// TwinCAT 3 PLC project PLC
// ProgramVersion: 3.1.4024.0
// libraries:
//   EfficientIO Energy Basic, * (EfficientIO)
//   Lynus Persistent Data V1, * (Lynus AG)
//   Lynus Standards, * (EfficientIO)
//   Tc2_EtherCAT, * (Beckhoff Automation GmbH)
//   Tc2_Standard, * (Beckhoff Automation GmbH)
//   Tc2_System, * (Beckhoff Automation GmbH)
//   Tc2_Utilities, * (Beckhoff Automation GmbH)
//   Tc3_Module, * (Beckhoff Automation GmbH)
// project tree:
//   FBs/EL3443_DPM/DUTs/ E_EL3443_DPM_Phase.TcDUT, E_EL3443_DPM_Total.TcDUT, MDP5001_341_7CD731EE.TcDUT (not stored), MDP5001_341_I_7CD731EE.TcDUT (not stored), MDP5001_341_O_7CD731EE.TcDUT (not stored), ST_EL3443_DPM_MUX_REAL.TcDUT (not stored), ST_EL3443_DPM_MUX_ULINT.TcDUT (not stored), ST_EL3443_DPM_StatusLx.TcDUT (not stored), ST_EL3443_DPM_StatusTotal.TcDUT (not stored), ST_EL3443_DPM_VariantLx.TcDUT (not stored), ST_EL3443_DPM_VariantTotal.TcDUT, ST_EL3443_DPM_VariantValues.TcDUT (not stored)
//   FBs/EL3443_DPM/ FB_EL3443_DPM.TcPOU (not stored)
//   FBs/EL3446 FW02 or higher/DUTs/ E_EL3446_Phase.TcDUT (not stored), MDP5001_342_066CA8C6.TcDUT (not stored), MDP5001_342_I_066CA8C6.TcDUT (not stored), MDP5001_342_O_066CA8C6.TcDUT (not stored), ST_EL3446_MUX_REAL.TcDUT (not stored), ST_EL3446_MUX_ULINT.TcDUT (not stored), ST_EL3446_StatusIx.TcDUT (not stored), ST_EL3446_VariantIx.TcDUT (not stored), ST_EL3446_VariantValues.TcDUT (not stored)
//   FBs/EL3446 FW02 or higher/ FB_EL3446.TcPOU (not stored)
//   FBs/ FB_CoE_EL3443.TcPOU, FB_CoE_EL3446.TcPOU (not stored), FB_EM_Beckhoff_EL3443.TcPOU, FB_EM_Beckhoff_EL3446.TcPOU
//   / PlcTask.TcTTO
//   POUs/ prgEM.TcPOU, prgHW.TcPOU
// real-time tasks:
//   TASK PlcTask: cycle T#10ms, priority 20, ADS port 350
// I/O:
//   DEVICE Gerät 2 (EtherCAT), AmsNetId 5.146.127.90.3.1
//     Klemme 1 (EK1200) [EK1200-5000 EtherCAT Netzteil (2A E-Bus)]
//       Klemme 2 (EL3443) [EL3443 3K. Leistungsmessung]
//       Klemme 3 (EL3446) [EL3446 DPM 6 K. Strommessklemme]
//       Klemme 4 (EL9011) [EL9011 Endklemme]
// variable links:
//   PLC/PLC Instance <-> Device 2 (EtherCAT)/Term 1 (EK1200)/Term 2 (EL3443)
//     PlcTask Inputs/prgHW.MDP5001_341_DPM_Data_Data_{1..20} <-> DPM Data/Data {1..20}  (20 links)
//     PlcTask Inputs/prgHW.MDP5001_341_L1_Basic_Current <-> L1 Basic/Current
//     PlcTask Inputs/prgHW.MDP5001_341_L2_Basic_Current <-> L2 Basic/Current
//     PlcTask Inputs/prgHW.MDP5001_341_L3_Basic_Current <-> L3 Basic/Current
//     PlcTask Inputs/prgHW.MDP5001_341_L1_Basic_Voltage <-> L1 Basic/Voltage
//     PlcTask Inputs/prgHW.MDP5001_341_L2_Basic_Voltage <-> L2 Basic/Voltage
//     PlcTask Inputs/prgHW.MDP5001_341_L3_Basic_Voltage <-> L3 Basic/Voltage
//     PlcTask Inputs/prgHW.MDP5001_341_L1_Power_Active_Power <-> L1 Power/Active Power
//     PlcTask Inputs/prgHW.MDP5001_341_L2_Power_Active_Power <-> L2 Power/Active Power
//     PlcTask Inputs/prgHW.MDP5001_341_L3_Power_Active_Power <-> L3 Power/Active Power
//     PlcTask Inputs/prgHW.MDP5001_341_L1_Power_Apparent_Power <-> L1 Power/Apparent Power
//     PlcTask Inputs/prgHW.MDP5001_341_L2_Power_Apparent_Power <-> L2 Power/Apparent Power
//     PlcTask Inputs/prgHW.MDP5001_341_L3_Power_Apparent_Power <-> L3 Power/Apparent Power
//     PlcTask Inputs/prgHW.MDP5001_341_L1_Power_Power_Factor <-> L1 Power/Power Factor
//     PlcTask Inputs/prgHW.MDP5001_341_L2_Power_Power_Factor <-> L2 Power/Power Factor
//     PlcTask Inputs/prgHW.MDP5001_341_L3_Power_Power_Factor <-> L3 Power/Power Factor
//     PlcTask Inputs/prgHW.MDP5001_341_L1_Power_Reactive_Power <-> L1 Power/Reactive Power
//     PlcTask Inputs/prgHW.MDP5001_341_L2_Power_Reactive_Power <-> L2 Power/Reactive Power
//     PlcTask Inputs/prgHW.MDP5001_341_L3_Power_Reactive_Power <-> L3 Power/Reactive Power
//     PlcTask Inputs/prgHW.MDP5001_341_L1_Status_Current_Guard_Error <-> L1 Status/Current Guard Error
//     PlcTask Inputs/prgHW.MDP5001_341_L2_Status_Current_Guard_Error <-> L2 Status/Current Guard Error
//     PlcTask Inputs/prgHW.MDP5001_341_L3_Status_Current_Guard_Error <-> L3 Status/Current Guard Error
//     PlcTask Inputs/prgHW.MDP5001_341_L1_Status_Current_Guard_Warning <-> L1 Status/Current Guard Warning
//     PlcTask Inputs/prgHW.MDP5001_341_L2_Status_Current_Guard_Warning <-> L2 Status/Current Guard Warning
//     PlcTask Inputs/prgHW.MDP5001_341_L3_Status_Current_Guard_Warning <-> L3 Status/Current Guard Warning
//     PlcTask Inputs/prgHW.MDP5001_341_L1_Status_Inaccurate_Current <-> L1 Status/Inaccurate Current
//     PlcTask Inputs/prgHW.MDP5001_341_L2_Status_Inaccurate_Current <-> L2 Status/Inaccurate Current
//     PlcTask Inputs/prgHW.MDP5001_341_L3_Status_Inaccurate_Current <-> L3 Status/Inaccurate Current
//     PlcTask Inputs/prgHW.MDP5001_341_L1_Status_Inaccurate_Voltage <-> L1 Status/Inaccurate Voltage
//     PlcTask Inputs/prgHW.MDP5001_341_L2_Status_Inaccurate_Voltage <-> L2 Status/Inaccurate Voltage
//     PlcTask Inputs/prgHW.MDP5001_341_L3_Status_Inaccurate_Voltage <-> L3 Status/Inaccurate Voltage
//     PlcTask Inputs/prgHW.MDP5001_341_L1_Status_Overcurrent <-> L1 Status/Overcurrent
//     PlcTask Inputs/prgHW.MDP5001_341_L2_Status_Overcurrent <-> L2 Status/Overcurrent
//     PlcTask Inputs/prgHW.MDP5001_341_L3_Status_Overcurrent <-> L3 Status/Overcurrent
//     PlcTask Inputs/prgHW.MDP5001_341_L1_Status_Overvoltage <-> L1 Status/Overvoltage
//     PlcTask Inputs/prgHW.MDP5001_341_L2_Status_Overvoltage <-> L2 Status/Overvoltage
//     PlcTask Inputs/prgHW.MDP5001_341_L3_Status_Overvoltage <-> L3 Status/Overvoltage
//     PlcTask Inputs/prgHW.MDP5001_341_L1_Status_TxPDO_Toggle <-> L1 Status/TxPDO Toggle
//     PlcTask Inputs/prgHW.MDP5001_341_L2_Status_TxPDO_Toggle <-> L2 Status/TxPDO Toggle
//     PlcTask Inputs/prgHW.MDP5001_341_L3_Status_TxPDO_Toggle <-> L3 Status/TxPDO Toggle
//     PlcTask Inputs/prgHW.MDP5001_341_L1_Status_Voltage_Guard_Error <-> L1 Status/Voltage Guard Error
//     PlcTask Inputs/prgHW.MDP5001_341_L2_Status_Voltage_Guard_Error <-> L2 Status/Voltage Guard Error
//     PlcTask Inputs/prgHW.MDP5001_341_L3_Status_Voltage_Guard_Error <-> L3 Status/Voltage Guard Error
//     PlcTask Inputs/prgHW.MDP5001_341_L1_Status_Voltage_Guard_Warning <-> L1 Status/Voltage Guard Warning
//     PlcTask Inputs/prgHW.MDP5001_341_L2_Status_Voltage_Guard_Warning <-> L2 Status/Voltage Guard Warning
//     PlcTask Inputs/prgHW.MDP5001_341_L3_Status_Voltage_Guard_Warning <-> L3 Status/Voltage Guard Warning
//     PlcTask Inputs/prgHW.MDP5001_341_L1_Status_Voltage_Sign_Bit <-> L1 Status/Voltage Sign Bit
//     PlcTask Inputs/prgHW.MDP5001_341_L2_Status_Voltage_Sign_Bit <-> L2 Status/Voltage Sign Bit
//     PlcTask Inputs/prgHW.MDP5001_341_L3_Status_Voltage_Sign_Bit <-> L3 Status/Voltage Sign Bit
//     PlcTask Inputs/prgHW.MDP5001_341_Total_Basic_Calculated_Neutral_Line_Current <-> Total Basic/Calculated Neutral Line Current
//     PlcTask Inputs/prgHW.MDP5001_341_Total_Basic_Frequency <-> Total Basic/Frequency
//     PlcTask Inputs/prgHW.MDP5001_341_Total_Basic_Power_Factor <-> Total Basic/Power Factor
//     PlcTask Inputs/prgHW.MDP5001_341_Total_Status_Active_Power_Guard_Error <-> Total Status/Active Power Guard Error
//     PlcTask Inputs/prgHW.MDP5001_341_Total_Status_Active_Power_Guard_Warning <-> Total Status/Active Power Guard Warning
//     PlcTask Inputs/prgHW.MDP5001_341_Total_Status_Apparent_Power_Guard_Error <-> Total Status/Apparent Power Guard Error
//     PlcTask Inputs/prgHW.MDP5001_341_Total_Status_Apparent_Power_Guard_Warning <-> Total Status/Apparent Power Guard Warning
//     PlcTask Inputs/prgHW.MDP5001_341_Total_Status_Frequency_Guard_Error <-> Total Status/Frequency Guard Error
//     PlcTask Inputs/prgHW.MDP5001_341_Total_Status_Frequency_Guard_Warning <-> Total Status/Frequency Guard Warning
//     PlcTask Inputs/prgHW.MDP5001_341_Total_Status_Grid_Direction <-> Total Status/Grid Direction
//     PlcTask Inputs/prgHW.MDP5001_341_Total_Status_Neutral_Current_Guard_Error <-> Total Status/Neutral Current Guard Error
//     PlcTask Inputs/prgHW.MDP5001_341_Total_Status_Neutral_Current_Guard_Warning <-> Total Status/Neutral Current Guard Warning
//     PlcTask Inputs/prgHW.MDP5001_341_Total_Status_Power_Quality_Factor <-> Total Status/Power Quality Factor
//     PlcTask Inputs/prgHW.MDP5001_341_Total_Status_Power_Quality_Guard_Error <-> Total Status/Power Quality Guard Error
//     PlcTask Inputs/prgHW.MDP5001_341_Total_Status_Power_Quality_Guard_Warning <-> Total Status/Power Quality Guard Warning
//     PlcTask Inputs/prgHW.MDP5001_341_Total_Status_System_State <-> Total Status/System State
//     PlcTask Inputs/prgHW.MDP5001_341_Total_Status_TxPDO_State <-> Total Status/TxPDO State
//     PlcTask Inputs/prgHW.MDP5001_341_Total_Status_TxPDO_Toggle <-> Total Status/TxPDO Toggle
//     PlcTask Inputs/prgHW.MDP5001_341_Total_Variant_Value_In_Index_1_REAL <-> Total Variant Value In/Index 1 REAL
//     PlcTask Inputs/prgHW.MDP5001_341_Total_Variant_Value_In_Index_2_REAL <-> Total Variant Value In/Index 2 REAL
//     PlcTask Inputs/prgHW.MDP5001_341_Total_Variant_Value_In_Index_3_REAL <-> Total Variant Value In/Index 3 REAL
//     PlcTask Inputs/prgHW.MDP5001_341_Total_Variant_Value_In_Index_4_ULINT <-> Total Variant Value In/Index 4 ULINT
//     PlcTask Inputs/prgHW.MDP5001_341_Total_Variant_Value_In_TxPDO_Toggle <-> Total Variant Value In/TxPDO Toggle
//     PlcTask Inputs/prgHW.MDP5001_341_Total_Variant_Value_In_Value_1_REAL <-> Total Variant Value In/Value 1 REAL
//     PlcTask Inputs/prgHW.MDP5001_341_Total_Variant_Value_In_Value_2_REAL <-> Total Variant Value In/Value 2 REAL
//     PlcTask Inputs/prgHW.MDP5001_341_Total_Variant_Value_In_Value_3_REAL <-> Total Variant Value In/Value 3 REAL
//     PlcTask Inputs/prgHW.MDP5001_341_Total_Variant_Value_In_Value_4_ULINT <-> Total Variant Value In/Value 4 ULINT
//     PlcTask Outputs/prgHW.MDP5001_341_Total_Interval_Reset_Interval <-> Total Interval/Reset Interval
//     PlcTask Outputs/prgHW.MDP5001_341_Total_Variant_Value_Out_Index_1_REAL <-> Total Variant Value Out/Index 1 REAL
//     PlcTask Outputs/prgHW.MDP5001_341_Total_Variant_Value_Out_Index_2_REAL <-> Total Variant Value Out/Index 2 REAL
//     PlcTask Outputs/prgHW.MDP5001_341_Total_Variant_Value_Out_Index_3_REAL <-> Total Variant Value Out/Index 3 REAL
//     PlcTask Outputs/prgHW.MDP5001_341_Total_Variant_Value_Out_Index_4_ULINT <-> Total Variant Value Out/Index 4 ULINT
//   PLC/PLC Instance <-> Device 2 (EtherCAT)/Term 1 (EK1200)/Term 3 (EL3446)
//     PlcTask Inputs/prgHW.MDP5001_342_DPM_Variant_Value_In_Index_1_REAL_1 <-> DPM Variant Value In/Index 1 REAL
//     PlcTask Inputs/prgHW.MDP5001_342_DPM_Variant_Value_In_Index_2_REAL_1 <-> DPM Variant Value In/Index 2 REAL
//     PlcTask Inputs/prgHW.MDP5001_342_DPM_Variant_Value_In_Index_3_REAL_1 <-> DPM Variant Value In/Index 3 REAL
//     PlcTask Inputs/prgHW.MDP5001_342_DPM_Variant_Value_In_Index_4_ULINT_1 <-> DPM Variant Value In/Index 4 ULINT
//     PlcTask Inputs/prgHW.MDP5001_342_DPM_Variant_Value_In_TxPDO_Toggle_1 <-> DPM Variant Value In/TxPDO Toggle
//     PlcTask Inputs/prgHW.MDP5001_342_DPM_Variant_Value_In_Value_1_REAL_1 <-> DPM Variant Value In/Value 1 REAL
//     PlcTask Inputs/prgHW.MDP5001_342_DPM_Variant_Value_In_Value_2_REAL_1 <-> DPM Variant Value In/Value 2 REAL
//     PlcTask Inputs/prgHW.MDP5001_342_DPM_Variant_Value_In_Value_3_REAL_1 <-> DPM Variant Value In/Value 3 REAL
//     PlcTask Inputs/prgHW.MDP5001_342_DPM_Variant_Value_In_Value_4_ULINT_1 <-> DPM Variant Value In/Value 4 ULINT
//     PlcTask Inputs/prgHW.MDP5001_342_I{1..6}_Channel_Active_Energy_1 <-> I{1..6} Channel/Active Energy  (6 links)
//     PlcTask Inputs/prgHW.MDP5001_342_I{1..6}_Channel_Active_Power_1 <-> I{1..6} Channel/Active Power  (6 links)
//     PlcTask Inputs/prgHW.MDP5001_342_I{1..6}_Channel_Active_Power_Guard_Error_1 <-> I{1..6} Channel/Active Power Guard Error  (6 links)
//     PlcTask Inputs/prgHW.MDP5001_342_I{1..6}_Channel_Active_Power_Guard_Warning_1 <-> I{1..6} Channel/Active Power Guard Warning  (6 links)
//     PlcTask Inputs/prgHW.MDP5001_342_I{1..6}_Channel_Apparent_Power_1 <-> I{1..6} Channel/Apparent Power  (6 links)
//     PlcTask Inputs/prgHW.MDP5001_342_I{1..6}_Channel_Apparent_Power_Guard_Error_1 <-> I{1..6} Channel/Apparent Power Guard Error  (6 links)
//     PlcTask Inputs/prgHW.MDP5001_342_I{1..6}_Channel_Apparent_Power_Guard_Warning_1 <-> I{1..6} Channel/Apparent Power Guard Warning  (6 links)
//     PlcTask Inputs/prgHW.MDP5001_342_I{1..6}_Channel_Current_1 <-> I{1..6} Channel/Current  (6 links)
//     PlcTask Inputs/prgHW.MDP5001_342_I{1..6}_Channel_Current_Guard_Error_1 <-> I{1..6} Channel/Current Guard Error  (6 links)
//     PlcTask Inputs/prgHW.MDP5001_342_I{1..6}_Channel_Current_Guard_Warning_1 <-> I{1..6} Channel/Current Guard Warning  (6 links)
//     PlcTask Inputs/prgHW.MDP5001_342_I{1..6}_Channel_DPM_Inaccurate_1 <-> I{1..6} Channel/DPM Inaccurate  (6 links)
//     PlcTask Inputs/prgHW.MDP5001_342_I{1..6}_Channel_DPM_Timeout_1 <-> I{1..6} Channel/DPM Timeout  (6 links)
//     PlcTask Inputs/prgHW.MDP5001_342_I{1..6}_Channel_Inaccurate_Current_1 <-> I{1..6} Channel/Inaccurate Current  (6 links)
//     PlcTask Inputs/prgHW.MDP5001_342_I{1..6}_Channel_Overcurrent_1 <-> I{1..6} Channel/Overcurrent  (6 links)
//     PlcTask Inputs/prgHW.MDP5001_342_I{1..6}_Channel_Reactive_Power_Fundamental_1 <-> I{1..6} Channel/Reactive Power Fundamental  (6 links)
//     PlcTask Inputs/prgHW.MDP5001_342_I{1..6}_Channel_Reactive_Power_Guard_Error_1 <-> I{1..6} Channel/Reactive Power Guard Error  (6 links)
//     PlcTask Inputs/prgHW.MDP5001_342_I{1..6}_Channel_Reactive_Power_Guard_Warning_1 <-> I{1..6} Channel/Reactive Power Guard Warning  (6 links)
//     PlcTask Inputs/prgHW.MDP5001_342_I{1..6}_Channel_TxPDO_Toggle_1 <-> I{1..6} Channel/TxPDO Toggle  (6 links)
//     PlcTask Outputs/prgHW.MDP5001_342_DPM_Data_Data_{1..20}_1 <-> DPM Data/Data {1..20}  (20 links)
//     PlcTask Outputs/prgHW.MDP5001_342_DPM_Variant_Value_Out_Index_1_REAL_1 <-> DPM Variant Value Out/Index 1 REAL
//     PlcTask Outputs/prgHW.MDP5001_342_DPM_Variant_Value_Out_Index_2_REAL_1 <-> DPM Variant Value Out/Index 2 REAL
//     PlcTask Outputs/prgHW.MDP5001_342_DPM_Variant_Value_Out_Index_3_REAL_1 <-> DPM Variant Value Out/Index 3 REAL
//     PlcTask Outputs/prgHW.MDP5001_342_DPM_Variant_Value_Out_Index_4_ULINT_1 <-> DPM Variant Value Out/Index 4 ULINT

CONFIGURATION PLC
    RESOURCE PLC ON TwinCAT3
        TASK PlcTask(INTERVAL := T#10ms, PRIORITY := 20);
        PROGRAM prgEM WITH PlcTask : prgEM;
        PROGRAM prgHW WITH PlcTask : prgHW;
    END_RESOURCE
END_CONFIGURATION

// ---- FBs/EL3443_DPM/DUTs/E_EL3443_DPM_Phase.TcDUT
(*This enum is equivalent to the selectors from the documentation " Confirmation of variable output values 1 - 4"*)
{attribute 'qualified_only'}
TYPE E_EL3443_DPM_Phase :
(
    nPhaseL1_OFFSET := 256,      //Offset Channel 1(Phase L1). The offset is added to the base selector     
    nPhaseL2_OFFSET := 512,      //Offset Channel 2(Phase L2). The offset is added to the base selector
    nPhaseL3_OFFSET := 768,      //Offset Channel 3(Phase L3). The offset is added to the base selector
    
    U_RMS := 1,                  // [V] (Real Selector: 1 (Examp.: 257 = 1 + 256 for ch. 1)) RMS value of the voltage
    U_peak := 2,                 // [V] (Real Selector: 2 (Examp.: 770 = 2 + 768 for ch. 3)) Peak value of the instantaneous voltage in the last interval
    U_Last_Zero_Cross := 3,      // [V] (UINT Selector: 3) DC time of the penultimate voltage zero crossing
    U_RMS_Minimum := 4,          // [V] (Real Selector: 4) Minimum RMS value of the voltage in the last interval
    U_RMS_Maximum := 5,          // [V] (Real Selector: 5) Maximum RMS value of the voltage in the last interval
    ULL := 6,                    // [V] (Real Selector: 6) RMS value of the phase-to-phase voltage (Channel 1: U_L1L2; Channel 1: U_L2L3; Channel 3: U_L3L1) 
    I_RMS := 8,                  // [A] (Real Selector: 8) RMS value of the current
    I_peak := 9,                 // [A] (Real Selector: 9) Peak value of the instantaneous current in the last interval
    I_RMS_Minimum := 11,         // [A] (Real Selector: 11) Minimum RMS value of the current in the last interval
    I_RMS_Maximum := 12,         // [A] (Real Selector: 12) Maximum RMS value of the current in the last interval
    Frequency := 17,             // [Hz] (Real Selector: 17) Frequency of this phase
    Phi := 21,                   // [°] (Real Selector: 21) Phase angle of the fundamental wave
    Cos_phi := 22,               // [-] (Real Selector: 22) Cosine of the fundamental wave phase angle
    Power_Factor := 23,          // [-] (Real Selector: 23) Power factor
    P := 26,                     // [W] (Real Selector: 26) Active power
    Pavg := 27,                  // [W] (Real Selector: 27) Average active power during the last interval
    Pmin := 28,                  // [W] (Real Selector: 28) Minimum active power in the last interval
    Pmax := 29,                  // [W] (Real Selector: 29) Maximum active power in the last interval
    S_ := 32,                    // [VA] (Real Selector: 32) Apparent power
    Savg := 33,                  // [VA] (Real Selector: 33) Average apparent power during the last interval
    Smin := 34,                  // [VA] (Real Selector: 34) Minimum apparent power in last interval
    Smax := 35,                  // [VA] (Real Selector: 35) Minimum apparent power in last interval
    Q := 38,                     // [Var] (Real Selector: 38) Reactive power
    Qavg := 39,                  // [Var] (Real Selector: 39) Average reactive power average during the last interval
    Qmin := 40,                  // [Var] (Real Selector: 40) Minimum reactive power in the last interval
    Qmax := 41,                  // [Var] (Real Selector: 41) Maximum reactive power in the last interval
    EP := 45,                    // [mhW] (UINT Selector: 45) Recorded active energy
    EP_pos := 46,                // [mhW] (UINT Selector: 46) Received active energy
    EP_neg := 47,                // [mhW] (UINT Selector: 47) Supplied active energy
	EP_interval := 48, 			// [mhW] (UINT Selector: 48) Recorded active energy in the last interval
	EP_pos_interval := 49, 		// [mhW] (UINT Selector: 49) Received active energy in the last interval
	EP_neg_interval := 50, 		// [mhW] (UINT Selector: 50) Supplied active energy in the last interval
    ES := 51,                    // [mhW] (UINT Selector: 51) Apparent energy
    ES_pos := 52,                // [mhW] (UINT Selector: 52) Apparent energy
    ES_neg := 53,                // [mhW] (UINT Selector: 53) Apparent energy
	ES_interval := 54, 			// [mhW] (UINT Selector: 54) Apparent energy in the last interval
	ES_pos_interval := 55, 		// [mhW] (UINT Selector: 55) Apparent energy in the last interval
	ES_neg_interval := 56, 		// [mhW] (UINT Selector: 56) Apparent energy in the last interval
    EQ_ := 57,                   // [mhW] (UINT Selector: 57) Reactive energy
    EQ_pos := 58,                // [mhW] (UINT Selector: 58) Reactive energy
    EQ_neg := 59,                // [mhW] (UINT Selector: 59) Reactive energy
	EQ_interval := 60, 			// [mhW] (UINT Selector: 60) Reactive energy in the last interval
	EQ_pos_interval := 61, 		// [mhW] (UINT Selector: 62) Reactive energy in the last interval
	EQ_neg_interval := 62, 		// [mhW] (UINT Selector: 63) Reactive energy in the last interval
    THD_U := 95,                 // [-] (Real Selector: 95) "Total Harmonic Distortion" is the distortion factor of the voltage. It indicates the ratio of the harmonic components of an oscillation relative to its fundamental.
    RMS_fund_U := 98,            // [V] (Real Selector: 98) Amplitude of the fundamental wave
    F_Ref_U := 99,               // [Hz] (Real Selector: 99) Reference frequency of the voltage harmonic: Specifies the underlying fundamental frequency, e.g.: 50 or 60 Hz.
    Harmonics_U := 100,          // [% of the fundamental wave] (Real Selector: 100-163) 0 => DC component, 1 => fundamental wave, 2=> 2nd harmonic, 3=> 3rd harmonic
    THD_I := 165,                // [-] (Real Selector: 165) "Total Harmonic Distortion" is the distortion factor of the current. It indicates the ratio of the harmonic components of an oscillation relative to its fundamental.
    TDD_I := 166,                // [% of the maximum current] (Real Selector: 166) "Total Demand Distortion" indicates the ratio between the current harmonics and the maximum current (EL3443: 1A and EL3443-0010: 5A)
    RMS_fund_I := 168,           // [A] (Real Selector: 168) Amplitude of the fundamental wave
    F_Ref_I := 169,              // [Hz] (Real Selector: 169) Reference frequency of the current harmonic: Specifies the underlying fundamental frequency, e.g.: 50 or 60 Hz.
    Harmonics_I := 170,          // [% of the fundamental wave] (Real Selector: 170-233) 0 => DC component, 1 => fundamental wave, 2=> 2nd harmonic, 3=> 3rd harmonic
    Error_INDEX_Not_Valid := 255 // [-] (Real Selector: 255) Error message: The selected index is not available.
)UINT;
END_TYPE

// ---- FBs/EL3443_DPM/DUTs/E_EL3443_DPM_Total.TcDUT
(*This enum is equivalent to the selectors from the documentation " Confirmation of variable output values 1 - 4"*)
{attribute 'qualified_only'}
TYPE E_EL3443_DPM_Total :
(
    nTotal_OFFSET := 1024,           // Offset for total values. The offset is added to the base selector
    
    In_RMS := 8,                     // [A]  (Real Selector: 1032 (= 1024 + 8))  Calculated RMS value of the neutral current
    Power_Factor := 23,              // [-]  (Real Selector: 1047 (= 1024 + 23))  Total power factor over all phases
    Ptot := 26,                      // [W]  (Real Selector: 1050 (= 1024 + 26))  Total active power
    Ptotavg := 27,                   // [W]  (Real Selector: 1051 (= 1024 + 27))  Average total active power during the last interval
    Ptotmin := 28,                   // [W]  (Real Selector: 1052 (= 1024 + 28))  Minimum total active power in the last interval
    Ptotmax := 29,                   // [W]  (Real Selector: 1053 (= 1024 + 29))  Maximum total active power in the last interval
    Stot := 32,                      // [VA]  (Real Selector: 1056 (= 1024 + 32))  Total apparent power
    Stotavg := 33,                   // [VA]  (Real Selector: 1057 (= 1024 + 33))  Average total apparent power during the last interval
    Stotmin := 34,                   // [VA]  (Real Selector: 1058 (= 1024 + 34))  Minimum total apparent power in the last interval
    Stotmax := 35,                   // [VA]  (Real Selector: 1059 (= 1024 + 35))  Maximum total apparent power in the last interval
    Qtot := 38,                      // [Var]  (Real Selector: 1062 (= 1024 + 38))  Total reactive power
    Qtotavg := 39,                   // [Var]  (Real Selector: 1063 (= 1024 + 39))  Average total reactive power during the last interval
    Qtotmin := 40,                   // [Var]  (Real Selector: 1064 (= 1024 + 40))  Minimum total reactive power in the last interval
    Qtotmax := 41,                   // [Var]  (Real Selector: 1065 (= 1024 + 41))  Maximum total reactive power in the last interval
    Eptot := 45,                     // [mWh]  (ULINT Selector: 1069 (= 1024 + 45))  Balanced total active energy
    EPtot_pos := 46,                 // [mWh]  (ULINT Selector: 1070 (= 1024 + 46))  Related total active energy
    EPtot_neg := 47,                 // [mWh]  (ULINT Selector: 1071 (= 1024 + 47))  Input total active energy
    Eptot_interval := 48,            // [mWh]  (ULINT Selector: 1072 (= 1024 + 48))  Balanced total active energy in last interval
    EPtot_pos_interval := 49,        // [mWh]  (ULINT Selector: 1073 (= 1024 + 49))  Total active energy related in the last interval
    EPtot_neg_interval := 50,        // [mWh]  (ULINT Selector: 1074 (= 1024 + 50))  Input total active energy the last interval
    EStot := 51,                     // [mWh]  (ULINT Selector: 1075 (= 1024 + 51))  Total apparent energy
    EStot_pos := 52,                 // [mWh]  (ULINT Selector: 1076 (= 1024 + 52))  Total apparent energy
    EStot_neg := 53,                 // [mWh]  (ULINT Selector: 1077 (= 1024 + 53))  Total apparent energy
    EStot_interval := 54,            // [mWh]  (ULINT Selector: 1078 (= 1024 + 54))  Total apparent energy in the last interval
    EStot_pos_interval := 55,        // [mWh]  (ULINT Selector: 1079 (= 1024 + 55))  Total apparent energy in the last interval
    EStot_neg_interval := 56,        // [mWh]  (ULINT Selector: 1080 (= 1024 + 56))  Total apparent energy in the last interval
    EQtot := 57,                     // [mWh]  (ULINT Selector: 1081 (= 1024 + 57))  Total reactive energy
    EQtot_pos := 58,                 // [mWh]  (ULINT Selector: 1082 (= 1024 + 58))  Total reactive energy
    EQtot_neg := 59,                 // [mWh]  (ULINT Selector: 1083 (= 1024 + 59))  Total reactive energy
    EQtot_interval := 60,            // [mWh]  (ULINT Selector: 1084 (= 1024 + 60))  Total reactive energy in the last interval
    EQtot_pos_interval := 61,        // [mWh]  (ULINT Selector: 1085 (= 1024 + 61))  Total reactive energy in the last interval
    EQtot_neg_interval := 62,        // [mWh]  (ULINT Selector: 1086 (= 1024 + 62))  Total reactive energy in the last interval
    PhiL1L2 := 70,                   // [°]  (Real Selector: 1094 (= 1024 + 70))  Phase shift angle between phase L1 and L2
    PhiL1L3 := 71,                   // [°]  (Real Selector: 1095 (= 1024 + 71))  Phase shift angle between phase L1 and L3
    Unbalance := 72,                 // [-]  (Real Selector: 1096 (= 1024 + 72))  Ratio between negative and positive voltage system
    PQF := 80,                       // [-]  (Real Selector: 1104 (= 1024 + 80))  Power quality factor
    PQF_Avg := 81,                   // [-]  (Real Selector: 1105 (= 1024 + 81))  Average value of the power quality factor during the last interval
    PQF_MIN := 82,                   // [-]  (Real Selector: 1106 (= 1024 + 82))  Minimum power quality factor in the last interval
    PQF_MAX := 83                    // [-]  (Real Selector: 1107 (= 1024 + 83))  Maximum power quality factor in the last interval
)UINT;      
END_TYPE

// ---- FBs/EL3443_DPM/DUTs/ST_EL3443_DPM_VariantTotal.TcDUT
TYPE ST_EL3443_DPM_VariantTotal :
STRUCT
    fIn_RMS : REAL; 			// [A]  (Real Selector: 1032 (= 1024 + 8))  Calculated RMS value of the neutral current
    fPower_Factor : REAL; 		// [-]  (Real Selector: 1047 (= 1024 + 23))  Total power factor over all phases
    fPtot : REAL; 				// [W]  (Real Selector: 1050 (= 1024 + 26))  Total active power
    fPtotavg : REAL; 			// [W]  (Real Selector: 1051 (= 1024 + 27))  Average total active power during the last interval
    fPtotmin : REAL; 			// [W]  (Real Selector: 1052 (= 1024 + 28))  Minimum total active power in the last interval
    fPtotmax : REAL; 			// [W]  (Real Selector: 1053 (= 1024 + 29))  Maximum total active power in the last interval
    fStot : REAL; 				// [VA]  (Real Selector: 1056 (= 1024 + 32))  Total apparent power
    fStotavg : REAL; 			// [VA]  (Real Selector: 1057 (= 1024 + 33))  Average total apparent power during the last interval
    fStotmin : REAL; 			// [VA]  (Real Selector: 1058 (= 1024 + 34))  Minimum total apparent power in the last interval
    fStotmax : REAL; 			// [VA]  (Real Selector: 1059 (= 1024 + 35))  Maximum total apparent power in the last interval
    fQtot : REAL; 				// [Var]  (Real Selector: 1062 (= 1024 + 38))  Total reactive power
    fQtotavg : REAL; 			// [Var]  (Real Selector: 1063 (= 1024 + 39))  Average total reactive power during the last interval
    fQtotmin : REAL; 			// [Var]  (Real Selector: 1064 (= 1024 + 40))  Minimum total reactive power in the last interval
    fQtotmax : REAL; 			// [Var]  (Real Selector: 1065 (= 1024 + 41))  Maximum total reactive power in the last interval
    nEptot : LINT; 				// [mWh]  (LINT Selector: 1069 (= 1024 + 45))  Balanced total active energy
    nEPtot_pos : ULINT; 		// [mWh]  (ULINT Selector: 1070 (= 1024 + 46))  Related total active energy
    nEPtot_neg : ULINT; 		// [mWh]  (ULINT Selector: 1071 (= 1024 + 47))  Input total active energy
    nEptot_interval : LINT; 	// [mWh]  (LINT Selector: 1072 (= 1024 + 48))  Balanced total active energy in last interval
    nEPtot_pos_interval : ULINT;// [mWh]  (ULINT Selector: 1073 (= 1024 + 49))  Total active energy related in the last interval
    nEPtot_neg_interval : ULINT;// [mWh]  (ULINT Selector: 1074 (= 1024 + 50))  Input total active energy the last interval
    nEStot : LINT; 				// [mWh]  (LINT Selector: 1075 (= 1024 + 51))  Total apparent energy
    nEStot_pos : ULINT; 		// [mWh]  (ULINT Selector: 1076 (= 1024 + 52))  Total apparent energy
    nEStot_neg : ULINT; 		// [mWh]  (ULINT Selector: 1077 (= 1024 + 53))  Total apparent energy
    nEStot_interval : LINT; 	// [mWh]  (LINT Selector: 1078 (= 1024 + 54))  Total apparent energy in the last interval
    nEStot_pos_interval : ULINT;// [mWh]  (ULINT Selector: 1079 (= 1024 + 55))  Total apparent energy in the last interval
    nEStot_neg_interval : ULINT;// [mWh]  (ULINT Selector: 1080 (= 1024 + 56))  Total apparent energy in the last interval
    nEQtot : LINT; 				// [mWh]  (LINT Selector: 1081 (= 1024 + 57))  Total reactive energy
    nEQtot_pos : ULINT; 		// [mWh]  (ULINT Selector: 1082 (= 1024 + 58))  Total reactive energy
    nEQtot_neg : ULINT; 		// [mWh]  (ULINT Selector: 1083 (= 1024 + 59))  Total reactive energy
    nEQtot_interval : LINT; 	// [mWh]  (LINT Selector: 1084 (= 1024 + 60))  Total reactive energy in the last interval
    nEQtot_pos_interval : ULINT;// [mWh]  (ULINT Selector: 1085 (= 1024 + 61))  Total reactive energy in the last interval
    nEQtot_neg_interval : ULINT;// [mWh]  (ULINT Selector: 1086 (= 1024 + 62))  Total reactive energy in the last interval
    fPhiL1L2 : REAL; 			// [°]  (Real Selector: 1094 (= 1024 + 70))  Phase shift angle between phase L1 and L2
    fPhiL1L3 : REAL; 			// [°]  (Real Selector: 1095 (= 1024 + 71))  Phase shift angle between phase L1 and L3
    fUnbalance : REAL; 			// [-]  (Real Selector: 1096 (= 1024 + 72))  Ratio between negative and positive voltage system
    fPQF : REAL; 				// [-]  (Real Selector: 1104 (= 1024 + 80))  Power quality factor
    fPQF_Avg : REAL; 			// [-]  (Real Selector: 1105 (= 1024 + 81))  Average value of the power quality factor during the last interval
    fPQF_Min : REAL; 			// [-]  (Real Selector: 1106 (= 1024 + 82))  Minimum power quality factor in the last interval
    fPQF_Max : REAL; 			// [-]  (Real Selector: 1107 (= 1024 + 83))  Maximum power quality factor in the last interval
END_STRUCT
END_TYPE

// ---- POUs/prgEM.TcPOU
PROGRAM prgEM
VAR
	fbEL3443DPM 		: FB_EM_Beckhoff_EL3443;	//EL3443 | PDO Assignment "DPM" (DPM: Distributed Power Measurement) |3-phase power measurement terminal with extended functionality
	fb_EL3446_1			: FB_EM_Beckhoff_EL3446;
	lr_RealPower_Halle	: LREAL;						
	lr_ApparentPower_Halle: LREAL;						
	lr_ReactivePower_Halle: LREAL;						
	lr_Frequency_Halle	: LREAL;						
                                                        
	lr_Voltage_L1N		: LREAL;						
	lr_Voltage_L2N		: LREAL;						
	lr_Voltage_L3N		: LREAL;						
	lr_Voltage_L1L2		: LREAL;						
	lr_Voltage_L2L3		: LREAL;						
	lr_Voltage_L3L1		: LREAL;						
 	lr_Current_L1		: LREAL;						
	lr_Current_L2		: LREAL;						
	lr_Current_L3		: LREAL;						
	lr_Power_House		: LREAL;						
	lr_RealPower_Kran		: LREAL;	
	real_Array_Modbus_Data	AT%MB0 : ARRAY[0..49] OF REAL;

END_VAR
VAR_INPUT
	stEL3443_IO 						: MDP5001_341_7CD731EE;
	stEL3446_IO_1 						: MDP5001_342_066CA8C6; 
	stEL3446_IO_2 						: MDP5001_342_066CA8C6; 
END_VAR
VAR PERSISTENT
	lr_EnergyCounter_Halle	: LREAL;					
END_VAR

// grid measurement
fbEL3443DPM(
	bEnable 	:= TRUE, 
	bInvers_CH1 := FALSE, 
	bInvers_CH2	:= FALSE, 
	bInvers_CH3	:= FALSE, 
	uiCurrentTransformerRatio:= 300,		// two cables,300:1 CTs only over one cable 
	nSlaveAddr 	:= 1001,
	b_SubIndex	:= 2,
	stEL3443_IO := ,
	pDpmData=> , 
	stDataEMPower=> , 
	stDataEMCounter=> , 
	stDataEMPowerRealTime=> , 
	stDataEMCounterRealTime=> );
fbEL3443DPM.stEL3443_IO.MDP5001_341_Input := stEL3443_IO.MDP5001_341_Input;
stEL3443_IO.MDP5001_341_Output	:= fbEL3443DPM.stEL3443_IO.MDP5001_341_Output;
 	
lr_RealPower_Halle		:= fbEL3443DPM.stDataEMPower.lrPowerTotal; 	
lr_ApparentPower_Halle 	:= fbEL3443DPM.stDataEMPower.lrApparentPowerTotal;
lr_ReactivePower_Halle	:= fbEL3443DPM.stDataEMPower.lrReactivePowerTotal;
lr_Frequency_Halle		:= fbEL3443DPM.stDataEMPower.lrFrequency;
lr_Voltage_L1N			:= fbEL3443DPM.stDataEMPower.lrVoltageL1N;
lr_Voltage_L2N			:= fbEL3443DPM.stDataEMPower.lrVoltageL2N;
lr_Voltage_L3N			:= fbEL3443DPM.stDataEMPower.lrVoltageL3N;
lr_Voltage_L1L2			:= fbEL3443DPM.stDataEMPower.lrVoltageL1L2;
lr_Voltage_L2L3			:= fbEL3443DPM.stDataEMPower.lrVoltageL2L3;
lr_Voltage_L3L1			:= fbEL3443DPM.stDataEMPower.lrVoltageL3L1;
lr_EnergyCounter_Halle	:= fbEL3443DPM.stDataEMCounter.lrTotalCounterEnergy_Consumption;
lr_Current_L1			:= fbEL3443DPM.stDataEMPower.lrCurrentL1;
lr_Current_L2			:= fbEL3443DPM.stDataEMPower.lrCurrentL2;
lr_Current_L3			:= fbEL3443DPM.stDataEMPower.lrCurrentL3;
	 
fb_EL3446_1(
	bEnable:= TRUE , 
	bEnableVariantValues:= TRUE, 
	pDpmData:= fbEL3443DPM.pDpmData, 
	nSlaveAddr:= 1002, 
	b_SubIndex	:= 2,
	bInvers_CH1:= FALSE, 
	bInvers_CH2:= FALSE, 
	bInvers_CH3:= FALSE, 
	bInvers_CH4:= FALSE, 
	bInvers_CH5:= FALSE, 
	bInvers_CH6:= FALSE, 
	uiCurrentTransformerRatio_CH1:= 300, 
	uiCurrentTransformerRatio_CH2:= 300, 
	uiCurrentTransformerRatio_CH3:= 300, 
	uiCurrentTransformerRatio_CH4:= 300, 
	uiCurrentTransformerRatio_CH5:= 300, 
	uiCurrentTransformerRatio_CH6:= 300, 
	uiVoltagePhaseSelector_CH1:= , 
	uiVoltagePhaseSelector_CH2:= , 
	uiVoltagePhaseSelector_CH3:= , 
	uiVoltagePhaseSelector_CH4:= , 
	uiVoltagePhaseSelector_CH5:= , 
	uiVoltagePhaseSelector_CH6:= , 
	bEnable3PhaseCH13:= TRUE, 
	bEnable3PhaseCH46:= TRUE, 
	stDataEMPowerRealTime:= fbEL3443DPM.stDataEMPowerRealTime, 
	stEL3446_IO := ,
	stDataEMPower_CH1=> , 
	stDataEMCounter_CH1=> , 
	stDataEMPowerRealTime_CH1=> , 
	stDataEMCounterRealTime_CH1=> , 
	stDataEMPower_CH2=> , 
	stDataEMCounter_CH2=> , 
	stDataEMPowerRealTime_CH2=> , 
	stDataEMCounterRealTime_CH2=> , 
	stDataEMPower_CH3=> , 
	stDataEMCounter_CH3=> , 
	stDataEMPowerRealTime_CH3=> , 
	stDataEMCounterRealTime_CH3=> , 
	stDataEMPower_CH4=> , 
	stDataEMCounter_CH4=> , 
	stDataEMPowerRealTime_CH4=> , 
	stDataEMCounterRealTime_CH4=> , 
	stDataEMPower_CH5=> , 
	stDataEMCounter_CH5=> , 
	stDataEMPowerRealTime_CH5=> , 
	stDataEMCounterRealTime_CH5=> , 
	stDataEMPower_CH6=> , 
	stDataEMCounter_CH6=> , 
	stDataEMPowerRealTime_CH6=> , 
	stDataEMCounterRealTime_CH6=> );
fb_EL3446_1.stEL3446_IO.MDP5001_342_Input := stEL3446_IO_1.MDP5001_342_Input;
stEL3446_IO_1.MDP5001_342_Output := 	fb_EL3446_1.stEL3446_IO.MDP5001_342_Output;

lr_RealPower_Kran := fb_EL3446_1.stDataEMPower_CH1.lrPowerConsumption;

real_Array_Modbus_Data[0] 	:= 		INT_TO_REAL(REAL_TO_INT(LREAL_TO_REAL(lr_RealPower_Halle    *10)))/10 ;
real_Array_Modbus_Data[1] 	:= 		INT_TO_REAL(REAL_TO_INT(LREAL_TO_REAL(lr_ApparentPower_Halle*10)))/10 ;
real_Array_Modbus_Data[2] 	:= 		INT_TO_REAL(REAL_TO_INT(LREAL_TO_REAL(lr_ReactivePower_Halle*10)))/10 ;
real_Array_Modbus_Data[3] 	:= 		INT_TO_REAL(REAL_TO_INT(LREAL_TO_REAL(lr_Frequency_Halle    *10)))/10 ;
real_Array_Modbus_Data[4] 	:= 		INT_TO_REAL(REAL_TO_INT(LREAL_TO_REAL(lr_Voltage_L1N     	*10)))/10 ;
real_Array_Modbus_Data[5] 	:= 		INT_TO_REAL(REAL_TO_INT(LREAL_TO_REAL(lr_Voltage_L2N     	*10)))/10 ;
real_Array_Modbus_Data[6] 	:= 		INT_TO_REAL(REAL_TO_INT(LREAL_TO_REAL(lr_Voltage_L3N    	*10)))/10 ;
real_Array_Modbus_Data[7]	:=      INT_TO_REAL(REAL_TO_INT(LREAL_TO_REAL(lr_Voltage_L1L2		*10)))/10  ;
real_Array_Modbus_Data[8]	:=      INT_TO_REAL(REAL_TO_INT(LREAL_TO_REAL(lr_Voltage_L2L3		*10)))/10  ;
real_Array_Modbus_Data[9]	:=      INT_TO_REAL(REAL_TO_INT(LREAL_TO_REAL(lr_Voltage_L3L1		*10)))/10  ;
real_Array_Modbus_Data[10]	:=      INT_TO_REAL(REAL_TO_INT(LREAL_TO_REAL(lr_Current_L1		  	*10)))/10      ;
real_Array_Modbus_Data[11]	:=      INT_TO_REAL(REAL_TO_INT(LREAL_TO_REAL(lr_Current_L2		  	*10)))/10      ;
real_Array_Modbus_Data[12]	:=      INT_TO_REAL(REAL_TO_INT(LREAL_TO_REAL(lr_Current_L3		  	*10)))/10      ;
real_Array_Modbus_Data[13]	:=      INT_TO_REAL(REAL_TO_INT(LREAL_TO_REAL(lr_RealPower_Kran 	*10)))/10    ;

END_PROGRAM

// ---- FBs/FB_EM_Beckhoff_EL3443.TcPOU
FUNCTION_BLOCK FB_EM_Beckhoff_EL3443
VAR_INPUT
	bEnable							: BOOL;											//Enable the function
 	bInvers_CH1						: BOOL;											//Invert the Output data from Channel 1 
	bInvers_CH2						: BOOL;											//Invert the Output data from Channel 2 
	bInvers_CH3						: BOOL;											//Invert the Output data from Channel 3
	uiCurrentTransformerRatio		: UINT;											//Current Transformer Ratio  
	nSlaveAddr						: UINT;											//EtherCat Slave ID	
 	b_SubIndex						: BYTE;											//AmsNet ID Index, typically 2 or 3
	stEL3443_IO 						: MDP5001_341_7CD731EE;
END_VAR
VAR_OUTPUT
   	pDpmData 						: POINTER TO ARRAY[1..20] OF UDINT;
	stDataEMPower					: ST_ElectricMeter_Output_Power;				//Output structure with Data from Electric Meter (Power Data) 
	stDataEMCounter					: ST_ElectricMeter_Output_Counter;				//Output structure with Data from Electric Meter (Counter Data) 
	stDataEMPowerRealTime			: ST_ElectricMeter_Output_Power;				//Output structure with Data from Electric Meter (Power Data RealTime)
	stDataEMCounterRealTime			: ST_ElectricMeter_Output_Counter;				//Output structure with Data from Electric Meter (Counter Data RealTime) 
END_VAR
VAR
	fbEM							: FB_ElectricMeter;								//Electric Meter Function
	fbEnergyCounter					: FB_EnergyCounter;								//FB energy Counter, because the KL3403 has no nice logic for the Energy value
	fbEL3443DPM 					: FB_EL3443_DPM;
	
	fb_WriteCOE_EL3443	:FB_Coe_EL3443;	
	m_COE_Done: BOOL;
	uiCurrentTransformerRatio_old		: UINT;											//Current Transformer Ratio  
	f_trig_Busy: f_trig;

	
	timDissableFunctions			: TON;											//Timer to dissable the Function after Lynus_Standards.Constants_General.tTimeDissableLynusFunctions Days without connection to the Lynus Cloud
	timResetConnectionOnGVL			: TON;											//Timer to try reset the connection Flag on the GVL. (When somebody delete the Connection Function and make only a onlinechange)
	timSetCounterValues				: TON;											//Timer to set the counter values from the KL3403 Function to the EM Function
	arrPD							: ARRAY[1..7] OF FB_PersistentData_Number;		//Function to save persistent data
	byWaitInStep					: BYTE;											//Wait in Step before start to clean data on PLC
	iStateGVLData					: INT;											//State machine to handle the data on the GVL
	diCounterForGVL					: DINT;											//Counter to clean old data on GVL
	real_Multiplier_CH1: REAL;
	real_Multiplier_CH2: REAL;
	real_Multiplier_CH3: REAL;
END_VAR

//Creator : Stefan Lackner
//Company : EfficientIO
//Date : xx.09.2023
//Version : 1.0.0.0


//With this function is possible to read out all Information from a EL3446

//NOTE for diNr.....Designation => 
//_IN = Here Data come in from other Functions or go out to other functions about the GVL
//_OUT = Here Data go out to other functions about the GVL



(*-------------------------------------------------------------Service from Backend is ready and check the connection to backen for dissabel/enable Function---------------------------------------------------------------*)

//Try to reset the variable for connection on the GVL. When all is normal then the Lynus Mqtt connection function set this variable to true in the next cycle
//When we have no connection to the backend then after Lynus_Standards.Constants_General.tTimeDissableLynusFunctions days the Function is dissabled with all of his functionalities
timResetConnectionOnGVL(IN:= NOT timResetConnectionOnGVL.Q, PT:= T#1H, Q=> , ET=> );
IF timResetConnectionOnGVL.Q THEN 
	Lynus_Standards.GVL_Communicator.bStateConnectionToEnableFunctions := FALSE; 
END_IF
IF NOT Lynus_Standards.GVL_Communicator.bStateConnectionToEnableFunctions THEN 
	timDissableFunctions.IN := TRUE; 
ELSE 
	timDissableFunctions.IN := FALSE; 
END_IF  
timDissableFunctions(IN:= , PT:= Lynus_Standards.Constants_General.tTimeDissableLynusFunctions, Q=> , ET=> );

// limit inputs
uiCurrentTransformerRatio	 := LIMIT (1,uiCurrentTransformerRatio,10000);


(*----------------------------------------------------------------------------------------EL3446 Communication----------------------------------------------------------------------------------------------*)
// write CoE values for phase selector

IF 	NOT m_COE_Done OR 	uiCurrentTransformerRatio <> uiCurrentTransformerRatio_old THEN
	fb_WriteCOE_EL3443.m_start := TRUE;
	m_COE_Done := TRUE;
	 uiCurrentTransformerRatio_old := uiCurrentTransformerRatio;
END_IF
f_trig_Busy(CLK := fb_WriteCOE_EL3443.m_Busy );
IF f_trig_Busy.Q AND (fb_WriteCOE_EL3443.m_CoE_Write_done OR fb_WriteCOE_EL3443.m_Error) THEN 
	fb_WriteCOE_EL3443.m_start := FALSE;
END_IF

fb_WriteCOE_EL3443(
	m_start:= , 
	nSlaveAddr:= nSlaveAddr, 
	b_SubIndex:= b_SubIndex,
	uiCurrentTransformerRatio:= uiCurrentTransformerRatio, 
	m_Busy=> , 
	m_CoE_Write_done=> , 
	m_Error=> , 
	udint_GetAMSNetID_Error=> , 
	udint_WriteCoE_Error=> );



fbEL3443DPM(
	bEnable:= TRUE, 
	stEL3443_IO:= stEL3443_IO , 
	stStatusTotal=> , 
	stStatusPhase_L1=> , 
	stStatusPhase_L2=> , 
	stStatusPhase_L3=> , 
	stVariantValues=> , 
	pDpmData=> pDpmData, 
	bError=> );






//Invert the Output data, because it is possible that the current transformers have been mounted in different mounting positions.
IF NOT bInvers_CH1 THEN
	real_Multiplier_CH1 := 1;
ELSE
	real_Multiplier_CH1 := -1;
END_IF
IF NOT bInvers_CH2 THEN
	real_Multiplier_CH2 := 1;
ELSE
	real_Multiplier_CH2 := -1;
END_IF
IF NOT bInvers_CH3 THEN
	real_Multiplier_CH3 := 1;
ELSE
	real_Multiplier_CH3 := -1;
END_IF


//Function
fbEM(
	bEnable:= bEnable, 
	bError:= , 
	bEnableReadOutFunction:= FALSE, 
	bWriteWithDelay:= TRUE, 
	bPowerDataInvers:= FALSE,
	bReadOutDataDone:= timSetCounterValues.Q,
	iTimeReadOutInterval:= 0, 
	iErrorCode:= , 
	iWarningCode:= , 
	lrTotalCounterEnergy_Consumption:= fbEnergyCounter.lrTotalCounterEnergy_Consumption,
	lrTotalCounterEnergy_Production:= fbEnergyCounter.lrTotalCounterEnergy_Production, 
	lrCounterEnergyT1_Consumption:= fbEnergyCounter.lrCounterEnergyT1_Consumption,
	lrCounterEnergyT2_Consumption:= fbEnergyCounter.lrCounterEnergyT2_Consumption,
	lrCounterEnergyT1_Production:= fbEnergyCounter.lrCounterEnergyT1_Production, 
	lrCounterEnergyT2_Production:= fbEnergyCounter.lrCounterEnergyT2_Production, 
	lrCurrentL1:=  REAL_TO_LREAL(fbEL3443DPM.stEL3443_IO.MDP5001_341_Input.MDP5001_341_L1_Basic_Current ),
	lrVoltageL1N:= REAL_TO_LREAL(fbEL3443DPM.stEL3443_IO.MDP5001_341_Input.MDP5001_341_L1_Basic_Voltage), 
	lrVoltageL1L2:= REAL_TO_LREAL(fbEL3443DPM.stEL3443_IO.MDP5001_341_Input.MDP5001_341_L1_Basic_Voltage * 1.73), 
	lrPowerL1:= REAL_TO_LREAL(fbEL3443DPM.stEL3443_IO.MDP5001_341_Input.MDP5001_341_L1_Power_Active_Power * real_Multiplier_CH1), 
	lrCurrentL2:=  REAL_TO_LREAL(fbEL3443DPM.stEL3443_IO.MDP5001_341_Input.MDP5001_341_L2_Basic_Current),
	lrVoltageL2N:= REAL_TO_LREAL(fbEL3443DPM.stEL3443_IO.MDP5001_341_Input.MDP5001_341_L2_Basic_Voltage), 
	lrVoltageL2L3:= REAL_TO_LREAL(fbEL3443DPM.stEL3443_IO.MDP5001_341_Input.MDP5001_341_L2_Basic_Voltage * 1.73), 
	lrPowerL2:= REAL_TO_LREAL(fbEL3443DPM.stEL3443_IO.MDP5001_341_Input.MDP5001_341_L2_Power_Active_Power  * real_Multiplier_CH2),	
	lrCurrentL3:=  REAL_TO_LREAL(fbEL3443DPM.stEL3443_IO.MDP5001_341_Input.MDP5001_341_L3_Basic_Current),
	lrVoltageL3N:= REAL_TO_LREAL(fbEL3443DPM.stEL3443_IO.MDP5001_341_Input.MDP5001_341_L3_Basic_Voltage), 
	lrVoltageL3L1:= REAL_TO_LREAL(fbEL3443DPM.stEL3443_IO.MDP5001_341_Input.MDP5001_341_L3_Basic_Voltage * 1.73), 
	lrPowerL3:= REAL_TO_LREAL(fbEL3443DPM.stEL3443_IO.MDP5001_341_Input.MDP5001_341_L3_Power_Active_Power * real_Multiplier_CH3),	

	lrPowerTotal:= fbEM.lrPowerL1+fbEM.lrPowerL2+fbEM.lrPowerL3, 
	lrFrequency:= REAL_TO_LREAL(fbEL3443DPM.stEL3443_IO.MDP5001_341_Input.MDP5001_341_Total_Basic_Frequency), 
 	lrApparentPowerTotal:= REAL_TO_LREAL(fbEL3443DPM.stEL3443_IO.MDP5001_341_Input.MDP5001_341_L1_Power_Apparent_Power + fbEL3443DPM.stEL3443_IO.MDP5001_341_Input.MDP5001_341_L2_Power_Apparent_Power + fbEL3443DPM.stEL3443_IO.MDP5001_341_Input.MDP5001_341_L3_Power_Apparent_Power) ,
	lrReactivePowerTotal:= REAL_TO_LREAL(fbEL3443DPM.stEL3443_IO.MDP5001_341_Input.MDP5001_341_L1_Power_Reactive_Power + fbEL3443DPM.stEL3443_IO.MDP5001_341_Input.MDP5001_341_L2_Power_Reactive_Power + fbEL3443DPM.stEL3443_IO.MDP5001_341_Input.MDP5001_341_L3_Power_Reactive_Power) , 
	tTimDelayOutput:= T#5S, 
	stDataEMOutPower=> stDataEMPowerRealTime, 
	stDataEMOutPowerDelay=> stDataEMPower, 
	stDataEMOutCounter=> stDataEMCounterRealTime,
	stDataEMOutCounterDelay=> stDataEMCounter,
	bReadOutMeter=> );
(*----------------------------------------------------------------------------------------Energy Counter Function----------------------------------------------------------------------------------------------*)

fbEnergyCounter(
	byActiveTariff:= 1, 
	lrPowerInput:= (fbEM.lrPowerTotal) / 1000, 
	lrTotalCounterEnergy_Consumption=> , 
	lrTotalCounterEnergy_Production=> , 
	lrCounterEnergyT1_Consumption=> , 
	lrCounterEnergyT2_Consumption=> , 
	lrCounterEnergyT1_Production=> , 
	lrCounterEnergyT2_Production=> );
(*----------------------------------------------------------------------------------------Electric Meter Function----------------------------------------------------------------------------------------------*)

//Error
IF timDissableFunctions.Q THEN 
	fbEM.bWarning := TRUE; 
	fbEM.iWarningCode := 0; 
ELSE 
	fbEM.bWarning := FALSE; 
END_IF 
IF Lynus_Standards.GVL_Energy.stNumberOfDevices.diNumberOfElectricMeters > Constants_Energy.diMaxNumberOfElectricMeters THEN 
	fbEM.bError := TRUE; 
ELSE 
	fbEM.bError := FALSE; 
END_IF
IF Lynus_Standards.GVL_Energy.stNumberOfDevices.diNumberOfElectricMeters > Constants_Energy.diMaxNumberOfElectricMeters THEN 
	fbEM.iErrorCode := 1;
ELSE 
	fbEM.iErrorCode := 0;
END_IF

timSetCounterValues(IN:= bEnable AND NOT timSetCounterValues.Q, PT:= T#2S, Q=> , ET=> );

END_FUNCTION_BLOCK

// ---- FBs/FB_CoE_EL3443.TcPOU
FUNCTION_BLOCK FB_CoE_EL3443
VAR_INPUT
	m_start: BOOL;
	nSlaveAddr	:UINT;
	b_SubIndex	:BYTE;
	uiCurrentTransformerRatio		: UINT;											//CT Ratio
END_VAR
VAR_OUTPUT
	m_Busy: BOOL;
	m_CoE_Write_done: BOOL;
	m_Error: bool;
	udint_GetAMSNetID_Error: UDINT;
	udint_WriteCoE_Error: UDINT;
END_VAR
VAR
	i_State	:UINT:=1;
	fb_GetAMSNetID	:FB_GetLocalAmsNetId;
  	fb_coe_write          : FB_EcCoESdoWrite; // Function Block for writing in CoE


	r_trig_Start: R_trig;
	i_errorCount: INT;
	i_AMSNetID_ReadOut_Succesfull: INT;
	str_AMSNetID: STRING(30);
 	real_Value     : REAL ; (* variable to be written to the CoE Object *)
 	
	i_CoE_Write_Succesfull: INT;

	real_Current_Min_Warning 	: REAL	:=-100;
	real_Current_Min_Error 		: REAL	:=-120;
	real_Current_Max_Warning 	: REAL	:= 100;
	real_Current_Max_Error 		: REAL	:= 120;
	


END_VAR


r_trig_Start(Clk := m_start);
b_SubIndex := LIMIT (1,b_SubIndex,8);
CASE i_State OF
	1: 		// wait for start
	IF r_trig_Start.Q THEN
		i_State := i_State+1;
		m_CoE_Write_done := FALSE;
		m_Busy := TRUE;
		m_Error := FALSE;
	END_IF

	2:		// read out ams net ID	
	fb_GetAMSNetID.bExecute := TRUE;
	i_State := i_State+1;
	
	3: 		// wait for read out
	IF fb_GetAMSNetID.bBusy = FALSE AND NOT fb_GetAMSNetID.bError = TRUE THEN
		fb_GetAMSNetID.bExecute := FALSE;
		i_AMSNetID_ReadOut_Succesfull := i_AMSNetID_ReadOut_Succesfull+1;
		i_State := i_State+1;
	ELSIF fb_GetAMSNetID.bError = TRUE THEN
		fb_GetAMSNetID.bExecute := FALSE;
		i_State := 100;
	END_IF
	
	4: 		// read out AMS Net ID done, convert received data
	str_AMSNetID := concat(BYTE_TO_STRING(fb_GetAMSNetID.AddrBytes[0]),'.');
	str_AMSNetID := concat(str_AMSNetID,BYTE_TO_STRING(fb_GetAMSNetID.AddrBytes[1]));
	str_AMSNetID := concat(str_AMSNetID,'.');	
	str_AMSNetID := concat(str_AMSNetID,BYTE_TO_STRING(fb_GetAMSNetID.AddrBytes[2]));
	str_AMSNetID := concat(str_AMSNetID,'.');
	str_AMSNetID := concat(str_AMSNetID,BYTE_TO_STRING(fb_GetAMSNetID.AddrBytes[3]));
	str_AMSNetID := concat(str_AMSNetID,'.');
	str_AMSNetID := concat(str_AMSNetID,BYTE_TO_STRING(b_SubIndex));
	str_AMSNetID := concat(str_AMSNetID,'.1');
	
	i_State := 10;

	10: 	// write channel 1 
	fb_coe_write.bExecute 	:= TRUE;
	fb_coe_write.nIndex		:= 16#8000;
	fb_coe_write.nSubIndex	:= 16#12; 
	real_Value 			:= UINT_TO_REAL(uiCurrentTransformerRatio);
	fb_coe_write.pSrcBuf	:= ADR(real_Value);
	fb_coe_write.cbBufLen	:= SIZEOF(real_Value);
	i_State := i_State+1;
	
	11: 	// wait for done or error
	IF NOT fb_coe_write.bBusy AND NOT fb_coe_write.bError THEN
		fb_coe_write.bExecute 	:= FALSE;
		i_CoE_Write_Succesfull := i_CoE_Write_Succesfull+1;
		i_State := i_State+1;
	ELSIF fb_coe_write.bError THEN
		fb_coe_write.bExecute 	:= FALSE;
		i_State := 100;
	END_IF

	12:		// wait 
	i_State := 20;
	
	20: 	// write channel 2 
	fb_coe_write.bExecute 	:= TRUE;
	fb_coe_write.nIndex		:= 16#8010;
	fb_coe_write.nSubIndex	:= 16#12; 
	real_Value 			:= UINT_TO_REAL(uiCurrentTransformerRatio);
	fb_coe_write.pSrcBuf	:= ADR(real_Value);
	fb_coe_write.cbBufLen	:= SIZEOF(real_Value);
	i_State := i_State+1;
	
	21: 	// wait for done or error
	IF NOT fb_coe_write.bBusy AND NOT fb_coe_write.bError THEN
		fb_coe_write.bExecute 	:= FALSE;
		i_CoE_Write_Succesfull := i_CoE_Write_Succesfull+1;
		i_State := i_State+1;
	ELSIF fb_coe_write.bError THEN
		fb_coe_write.bExecute 	:= FALSE;
		i_State := 100;
	END_IF

	22:		// wait 
	i_State := 30;

	30: 	// write channel 3 
	fb_coe_write.bExecute 	:= TRUE;
	fb_coe_write.nIndex		:= 16#8020;
	fb_coe_write.nSubIndex	:= 16#12; 
	real_Value 			:= UINT_TO_REAL(uiCurrentTransformerRatio);
	fb_coe_write.pSrcBuf	:= ADR(real_Value);
	fb_coe_write.cbBufLen	:= SIZEOF(real_Value);
	i_State := i_State+1;
	
	31: 	// wait for done or error
	IF NOT fb_coe_write.bBusy AND NOT fb_coe_write.bError THEN
		fb_coe_write.bExecute 	:= FALSE;
		i_CoE_Write_Succesfull := i_CoE_Write_Succesfull+1;
		i_State := i_State+1;
	ELSIF fb_coe_write.bError THEN
		fb_coe_write.bExecute 	:= FALSE;
		i_State := 100;
	END_IF

	32:		// wait 
	i_State := 40;		

	40: 	// write Channel 1 current guard min error 
	fb_coe_write.bExecute 	:= TRUE;
	fb_coe_write.nIndex		:= 16#8001;
	fb_coe_write.nSubIndex	:= 16#15; 
	real_Value 			:= (real_Current_Min_Error);
	fb_coe_write.pSrcBuf	:= ADR(real_Value);
	fb_coe_write.cbBufLen	:= SIZEOF(real_Value);
	i_State := i_State+1;
	
	41: 	// wait for done or error
	IF NOT fb_coe_write.bBusy AND NOT fb_coe_write.bError THEN
		fb_coe_write.bExecute 	:= FALSE;
		i_CoE_Write_Succesfull := i_CoE_Write_Succesfull+1;
		i_State := i_State+1;
	ELSIF fb_coe_write.bError THEN
		fb_coe_write.bExecute 	:= FALSE;
		i_State := 100;
	END_IF
	
	42:		// wait 
	i_State := i_State+1;		

	43: 	// write Channel 1 current guard min warning 
	fb_coe_write.bExecute 	:= TRUE;
	fb_coe_write.nIndex		:= 16#8001;
	fb_coe_write.nSubIndex	:= 16#16; 
	real_Value 			:= (real_Current_Min_Warning);
	fb_coe_write.pSrcBuf	:= ADR(real_Value);
	fb_coe_write.cbBufLen	:= SIZEOF(real_Value);
	i_State := i_State+1;
	
	44: 	// wait for done or error
	IF NOT fb_coe_write.bBusy AND NOT fb_coe_write.bError THEN
		fb_coe_write.bExecute 	:= FALSE;
		i_CoE_Write_Succesfull := i_CoE_Write_Succesfull+1;
		i_State := i_State+1;
	ELSIF fb_coe_write.bError THEN
		fb_coe_write.bExecute 	:= FALSE;
		i_State := 100;
	END_IF

	45:		// wait 
	i_State := i_State+1;		

	46: 	// write Channel 1 current guard max warning 
	fb_coe_write.bExecute 	:= TRUE;
	fb_coe_write.nIndex		:= 16#8001;
	fb_coe_write.nSubIndex	:= 16#17; 
	real_Value 			:= (real_Current_Max_Warning);
	fb_coe_write.pSrcBuf	:= ADR(real_Value);
	fb_coe_write.cbBufLen	:= SIZEOF(real_Value);
	i_State := i_State+1;
	
	47: 	// wait for done or error
	IF NOT fb_coe_write.bBusy AND NOT fb_coe_write.bError THEN
		fb_coe_write.bExecute 	:= FALSE;
		i_CoE_Write_Succesfull := i_CoE_Write_Succesfull+1;
		i_State := i_State+1;
	ELSIF fb_coe_write.bError THEN
		fb_coe_write.bExecute 	:= FALSE;
		i_State := 100;
	END_IF
	
	48:		// wait 
	i_State := i_State+1;		

	49: 	// write Channel 1 current guard max error 
	fb_coe_write.bExecute 	:= TRUE;
	fb_coe_write.nIndex		:= 16#8001;
	fb_coe_write.nSubIndex	:= 16#18; 
	real_Value 			:= (real_Current_Max_Error);
	fb_coe_write.pSrcBuf	:= ADR(real_Value);
	fb_coe_write.cbBufLen	:= SIZEOF(real_Value);
	i_State := i_State+1;
	
	50: 	// wait for done or error
	IF NOT fb_coe_write.bBusy AND NOT fb_coe_write.bError THEN
		fb_coe_write.bExecute 	:= FALSE;
		i_CoE_Write_Succesfull := i_CoE_Write_Succesfull+1;
		i_State := i_State+1;
	ELSIF fb_coe_write.bError THEN
		fb_coe_write.bExecute 	:= FALSE;
		i_State := 100;
	END_IF

	51:		// wait 
	i_State := i_State+1;	

	52: 	// write Channel 2 current guard min error 
	fb_coe_write.bExecute 	:= TRUE;
	fb_coe_write.nIndex		:= 16#8011;
	fb_coe_write.nSubIndex	:= 16#15; 
	real_Value 			:= (real_Current_Min_Error);
	fb_coe_write.pSrcBuf	:= ADR(real_Value);
	fb_coe_write.cbBufLen	:= SIZEOF(real_Value);
	i_State := i_State+1;
	
	53: 	// wait for done or error
	IF NOT fb_coe_write.bBusy AND NOT fb_coe_write.bError THEN
		fb_coe_write.bExecute 	:= FALSE;
		i_CoE_Write_Succesfull := i_CoE_Write_Succesfull+1;
		i_State := i_State+1;
	ELSIF fb_coe_write.bError THEN
		fb_coe_write.bExecute 	:= FALSE;
		i_State := 100;
	END_IF
	
	54:		// wait 
	i_State := i_State+1;		

	55: 	// write Channel 2 current guard min warning 
	fb_coe_write.bExecute 	:= TRUE;
	fb_coe_write.nIndex		:= 16#8011;
	fb_coe_write.nSubIndex	:= 16#16; 
	real_Value 			:= (real_Current_Min_Warning);
	fb_coe_write.pSrcBuf	:= ADR(real_Value);
	fb_coe_write.cbBufLen	:= SIZEOF(real_Value);
	i_State := i_State+1;
	
	56: 	// wait for done or error
	IF NOT fb_coe_write.bBusy AND NOT fb_coe_write.bError THEN
		fb_coe_write.bExecute 	:= FALSE;
		i_CoE_Write_Succesfull := i_CoE_Write_Succesfull+1;
		i_State := i_State+1;
	ELSIF fb_coe_write.bError THEN
		fb_coe_write.bExecute 	:= FALSE;
		i_State := 100;
	END_IF

	57:		// wait 
	i_State := i_State+1;		

	58: 	// write Channel 2 current guard max warning 
	fb_coe_write.bExecute 	:= TRUE;
	fb_coe_write.nIndex		:= 16#8011;
	fb_coe_write.nSubIndex	:= 16#17; 
	real_Value 			:= (real_Current_Max_Warning);
	fb_coe_write.pSrcBuf	:= ADR(real_Value);
	fb_coe_write.cbBufLen	:= SIZEOF(real_Value);
	i_State := i_State+1;
	
	59: 	// wait for done or error
	IF NOT fb_coe_write.bBusy AND NOT fb_coe_write.bError THEN
		fb_coe_write.bExecute 	:= FALSE;
		i_CoE_Write_Succesfull := i_CoE_Write_Succesfull+1;
		i_State := i_State+1;
	ELSIF fb_coe_write.bError THEN
		fb_coe_write.bExecute 	:= FALSE;
		i_State := 100;
	END_IF
	
	60:		// wait 
	i_State := i_State+1;		

	61: 	// write Channel 2 current guard max error 
	fb_coe_write.bExecute 	:= TRUE;
	fb_coe_write.nIndex		:= 16#8011;
	fb_coe_write.nSubIndex	:= 16#18; 
	real_Value 			:= (real_Current_Max_Error);
	fb_coe_write.pSrcBuf	:= ADR(real_Value);
	fb_coe_write.cbBufLen	:= SIZEOF(real_Value);
	i_State := i_State+1;
	
	62: 	// wait for done or error
	IF NOT fb_coe_write.bBusy AND NOT fb_coe_write.bError THEN
		fb_coe_write.bExecute 	:= FALSE;
		i_CoE_Write_Succesfull := i_CoE_Write_Succesfull+1;
		i_State := i_State+1;
	ELSIF fb_coe_write.bError THEN
		fb_coe_write.bExecute 	:= FALSE;
		i_State := 100;
	END_IF
	
	63:		// wait 
	i_State := i_State+1;	

	64: 	// write Channel 3 current guard min error 
	fb_coe_write.bExecute 	:= TRUE;
	fb_coe_write.nIndex		:= 16#8021;
	fb_coe_write.nSubIndex	:= 16#15; 
	real_Value 			:= (real_Current_Min_Error);
	fb_coe_write.pSrcBuf	:= ADR(real_Value);
	fb_coe_write.cbBufLen	:= SIZEOF(real_Value);
	i_State := i_State+1;
	
	65: 	// wait for done or error
	IF NOT fb_coe_write.bBusy AND NOT fb_coe_write.bError THEN
		fb_coe_write.bExecute 	:= FALSE;
		i_CoE_Write_Succesfull := i_CoE_Write_Succesfull+1;
		i_State := i_State+1;
	ELSIF fb_coe_write.bError THEN
		fb_coe_write.bExecute 	:= FALSE;
		i_State := 100;
	END_IF
	
	66:		// wait 
	i_State := i_State+1;		

	67: 	// write Channel 3 current guard min warning 
	fb_coe_write.bExecute 	:= TRUE;
	fb_coe_write.nIndex		:= 16#8021;
	fb_coe_write.nSubIndex	:= 16#16; 
	real_Value 			:= (real_Current_Min_Warning);
	fb_coe_write.pSrcBuf	:= ADR(real_Value);
	fb_coe_write.cbBufLen	:= SIZEOF(real_Value);
	i_State := i_State+1;
	
	68: 	// wait for done or error
	IF NOT fb_coe_write.bBusy AND NOT fb_coe_write.bError THEN
		fb_coe_write.bExecute 	:= FALSE;
		i_CoE_Write_Succesfull := i_CoE_Write_Succesfull+1;
		i_State := i_State+1;
	ELSIF fb_coe_write.bError THEN
		fb_coe_write.bExecute 	:= FALSE;
		i_State := 100;
	END_IF

	69:		// wait 
	i_State := i_State+1;		

	70: 	// write Channel 3 current guard max warning 
	fb_coe_write.bExecute 	:= TRUE;
	fb_coe_write.nIndex		:= 16#8021;
	fb_coe_write.nSubIndex	:= 16#17; 
	real_Value 			:= (real_Current_Max_Warning);
	fb_coe_write.pSrcBuf	:= ADR(real_Value);
	fb_coe_write.cbBufLen	:= SIZEOF(real_Value);
	i_State := i_State+1;
	
	71: 	// wait for done or error
	IF NOT fb_coe_write.bBusy AND NOT fb_coe_write.bError THEN
		fb_coe_write.bExecute 	:= FALSE;
		i_CoE_Write_Succesfull := i_CoE_Write_Succesfull+1;
		i_State := i_State+1;
	ELSIF fb_coe_write.bError THEN
		fb_coe_write.bExecute 	:= FALSE;
		i_State := 100;
	END_IF
	
	72:		// wait 
	i_State := i_State+1;		

	73: 	// write Channel 3 current guard max warning 
	fb_coe_write.bExecute 	:= TRUE;
	fb_coe_write.nIndex		:= 16#8021;
	fb_coe_write.nSubIndex	:= 16#18; 
	real_Value 			:= (real_Current_Max_Error);
	fb_coe_write.pSrcBuf	:= ADR(real_Value);
	fb_coe_write.cbBufLen	:= SIZEOF(real_Value);
	i_State := i_State+1;
	
	74: 	// wait for done or error
	IF NOT fb_coe_write.bBusy AND NOT fb_coe_write.bError THEN
		fb_coe_write.bExecute 	:= FALSE;
		i_CoE_Write_Succesfull := i_CoE_Write_Succesfull+1;
		i_State := i_State+1;
	ELSIF fb_coe_write.bError THEN
		fb_coe_write.bExecute 	:= FALSE;
		i_State := 100;
	END_IF	
	
	75:		// wait *)
	m_CoE_Write_done := TRUE;
	m_Busy := FALSE;
	i_State := 1;	
	
	100: 	//error state
	i_errorCount := i_errorCount +1;
	udint_GetAMSNetID_Error := fb_GetAMSNetID.nErrId;
	udint_WriteCoE_Error := fb_coe_write.nErrId;
	m_Busy := FALSE;
	m_Error := true;
	i_State := 1;

END_CASE


fb_GetAMSNetID(
	bExecute:= , 
	tTimeOut:= T#2S, 
	bBusy=> , 
	bError=> , 
	nErrId=> , 
	AddrString=> , 
	AddrBytes=> );
	
fb_coe_write(
	sNetId:= str_AMSNetID, 
	nSlaveAddr:= nSlaveAddr, 
	nSubIndex:= , 
	nIndex:= , 
    pSrcBuf    := ,
    cbBufLen   := ,
	bExecute:= , 
	tTimeout:= T#2S , 
	bBusy=> , 
	bError=> , 
	nErrId=> );

END_FUNCTION_BLOCK

// ---- FBs/FB_EM_Beckhoff_EL3446.TcPOU
FUNCTION_BLOCK FB_EM_Beckhoff_EL3446
VAR_INPUT
	bEnable							: BOOL;											//Enable the function
  	bEnableVariantValues 			: BOOL; //Enables the Variant values to be queried using the multiplexer functions of the block
    pDpmData 						: POINTER TO ARRAY[1..20] OF UDINT;
	nSlaveAddr						: UINT;											//EtherCat Slave ID	
 	b_SubIndex						: BYTE;											//AmsNet ID Index, typically 2 or 3
 	bInvers_CH1						: BOOL;											//Invert the Output data from Channel 1 
	bInvers_CH2						: BOOL;											//Invert the Output data from Channel 2 
	bInvers_CH3						: BOOL;											//Invert the Output data from Channel 3
	bInvers_CH4						: BOOL;											//Invert the Output data from Channel 4
	bInvers_CH5						: BOOL;											//Invert the Output data from Channel 5
	bInvers_CH6						: BOOL;											//Invert the Output data from Channel 6
	uiCurrentTransformerRatio_CH1	: UINT;											//Current Transformer Ratio for Channel 1 
	uiCurrentTransformerRatio_CH2	: UINT;											//Current Transformer Ratio for Channel 2 
	uiCurrentTransformerRatio_CH3	: UINT;											//Current Transformer Ratio for Channel 3 
	uiCurrentTransformerRatio_CH4	: UINT;											//Current Transformer Ratio for Channel 4 
	uiCurrentTransformerRatio_CH5	: UINT;											//Current Transformer Ratio for Channel 5 
	uiCurrentTransformerRatio_CH6	: UINT;											//Current Transformer Ratio for Channel 6
	uiVoltagePhaseSelector_CH1		: UINT;											//Voltage Phase Selector 1/2/3 for Channel 1
	uiVoltagePhaseSelector_CH2		: UINT;											//Voltage Phase Selector 1/2/3 for Channel 2
	uiVoltagePhaseSelector_CH3		: UINT;											//Voltage Phase Selector 1/2/3 for Channel 3
	uiVoltagePhaseSelector_CH4		: UINT;											//Voltage Phase Selector 1/2/3 for Channel 4
	uiVoltagePhaseSelector_CH5		: UINT;											//Voltage Phase Selector 1/2/3 for Channel 5
	uiVoltagePhaseSelector_CH6		: UINT;											//Voltage Phase Selector 1/2/3 for Channel 6 
	bEnable3PhaseCH13				: BOOL;											//Enable 3 phase measurement Channel 1-3
	bEnable3PhaseCH46				: BOOL;											//Enable 3 phase measurement Channel 4-6
	stDataEMPowerRealTime			: ST_ElectricMeter_Output_Power;				//Output structure with Data from Electric Meter (Power Data RealTime) used adding voltage to output struct
    stEL3446_IO : MDP5001_342_066CA8C6; 
END_VAR
VAR_OUTPUT
	stDataEMPower_CH1				: ST_ElectricMeter_Output_Power;				//Output structure with Data from Electric Meter (Power Data) for Channel 1
	stDataEMCounter_CH1				: ST_ElectricMeter_Output_Counter;				//Output structure with Data from Electric Meter (Counter Data) for Channel 1
	stDataEMPowerRealTime_CH1		: ST_ElectricMeter_Output_Power;				//Output structure with Data from Electric Meter (Power Data RealTime) for Channel 1
	stDataEMCounterRealTime_CH1		: ST_ElectricMeter_Output_Counter;				//Output structure with Data from Electric Meter (Counter Data RealTime) for Channel 1

	stDataEMPower_CH2				: ST_ElectricMeter_Output_Power;				//Output structure with Data from Electric Meter (Power Data) for Channel 2
	stDataEMCounter_CH2				: ST_ElectricMeter_Output_Counter;				//Output structure with Data from Electric Meter (Counter Data) for Channel 2
	stDataEMPowerRealTime_CH2		: ST_ElectricMeter_Output_Power;				//Output structure with Data from Electric Meter (Power Data RealTime) for Channel 2
	stDataEMCounterRealTime_CH2		: ST_ElectricMeter_Output_Counter;				//Output structure with Data from Electric Meter (Counter Data RealTime) for Channel 2

	stDataEMPower_CH3				: ST_ElectricMeter_Output_Power;				//Output structure with Data from Electric Meter (Power Data) for Channel 3
	stDataEMCounter_CH3				: ST_ElectricMeter_Output_Counter;				//Output structure with Data from Electric Meter (Counter Data) for Channel 3
	stDataEMPowerRealTime_CH3		: ST_ElectricMeter_Output_Power;				//Output structure with Data from Electric Meter (Power Data RealTime) for Channel 3
	stDataEMCounterRealTime_CH3		: ST_ElectricMeter_Output_Counter;				//Output structure with Data from Electric Meter (Counter Data RealTime) for Channel 3

	stDataEMPower_CH4				: ST_ElectricMeter_Output_Power;				//Output structure with Data from Electric Meter (Power Data) for Channel 4
	stDataEMCounter_CH4				: ST_ElectricMeter_Output_Counter;				//Output structure with Data from Electric Meter (Counter Data) for Channel 4
	stDataEMPowerRealTime_CH4		: ST_ElectricMeter_Output_Power;				//Output structure with Data from Electric Meter (Power Data RealTime) for Channel 4
	stDataEMCounterRealTime_CH4		: ST_ElectricMeter_Output_Counter;				//Output structure with Data from Electric Meter (Counter Data RealTime) for Channel 4

	stDataEMPower_CH5				: ST_ElectricMeter_Output_Power;				//Output structure with Data from Electric Meter (Power Data) for Channel 5
	stDataEMCounter_CH5				: ST_ElectricMeter_Output_Counter;				//Output structure with Data from Electric Meter (Counter Data) for Channel 5
	stDataEMPowerRealTime_CH5		: ST_ElectricMeter_Output_Power;				//Output structure with Data from Electric Meter (Power Data RealTime) for Channel 5
	stDataEMCounterRealTime_CH5		: ST_ElectricMeter_Output_Counter;				//Output structure with Data from Electric Meter (Counter Data RealTime) for Channel 5

	stDataEMPower_CH6				: ST_ElectricMeter_Output_Power;				//Output structure with Data from Electric Meter (Power Data) for Channel 6
	stDataEMCounter_CH6				: ST_ElectricMeter_Output_Counter;				//Output structure with Data from Electric Meter (Counter Data) for Channel 6
	stDataEMPowerRealTime_CH6		: ST_ElectricMeter_Output_Power;				//Output structure with Data from Electric Meter (Power Data RealTime) for Channel 6
	stDataEMCounterRealTime_CH6		: ST_ElectricMeter_Output_Counter;				//Output structure with Data from Electric Meter (Counter Data RealTime) for Channel 6	
	
END_VAR
VAR
	fbEM_CH1						: FB_ElectricMeter;								//Electric Meter Function
	fbEnergyCounter_CH1				: FB_EnergyCounter;								//FB energy Counter, because the KL3403 has no nice logic for the Energy value
	fbEM_CH2						: FB_ElectricMeter;								//Electric Meter Function
	fbEnergyCounter_CH2				: FB_EnergyCounter;								//FB energy Counter, because the KL3403 has no nice logic for the Energy value
	fbEM_CH3						: FB_ElectricMeter;								//Electric Meter Function
	fbEnergyCounter_CH3				: FB_EnergyCounter;								//FB energy Counter, because the KL3403 has no nice logic for the Energy value
	fbEM_CH4						: FB_ElectricMeter;								//Electric Meter Function
	fbEnergyCounter_CH4				: FB_EnergyCounter;								//FB energy Counter, because the KL3403 has no nice logic for the Energy value
	fbEM_CH5						: FB_ElectricMeter;								//Electric Meter Function
	fbEnergyCounter_CH5				: FB_EnergyCounter;								//FB energy Counter, because the KL3403 has no nice logic for the Energy value
	fbEM_CH6						: FB_ElectricMeter;								//Electric Meter Function
	fbEnergyCounter_CH6				: FB_EnergyCounter;								//FB energy Counter, because the KL3403 has no nice logic for the Energy value
	fbEL3446_wEL3443	: FB_EL3446; 		//EL3446 | 6-channel current input terminal 1 A AC/DC for distributed power measurement (FW02 or higher) for DPM with EL3443
	
	timDissableFunctions			: TON;											//Timer to dissable the Function after Lynus_Standards.Constants_General.tTimeDissableLynusFunctions Days without connection to the Lynus Cloud
	timResetConnectionOnGVL			: TON;											//Timer to try reset the connection Flag on the GVL. (When somebody delete the Connection Function and make only a onlinechange)
	timSetCounterValues				: TON;											//Timer to set the counter values from the KL3403 Function to the EM Function
	arrPD							: ARRAY[1..7] OF FB_PersistentData_Number;		//Function to save persistent data
	byWaitInStep					: BYTE;											//Wait in Step before start to clean data on PLC
	iStateGVLData					: INT;											//State machine to handle the data on the GVL
	diCounterForGVL					: DINT;											//Counter to clean old data on GVL
	bInit: BOOL;
	m_COE_Done: BOOL;
	FB_CoE_EL3446 :FB_CoE_EL3446;
	uiVoltagePhaseSelector_old_CH1		: UINT;											
	uiVoltagePhaseSelector_old_CH2		: UINT;											
	uiVoltagePhaseSelector_old_CH3		: UINT;											
	uiVoltagePhaseSelector_old_CH4		: UINT;											
	uiVoltagePhaseSelector_old_CH5		: UINT;											
	uiVoltagePhaseSelector_old_CH6		: UINT;											
	
	f_trig_Busy: f_trig;

	real_Multiplier_CH1: REAL;
	real_Multiplier_CH2: REAL;
	real_Multiplier_CH3: REAL;
	real_Multiplier_CH4: REAL;
	real_Multiplier_CH5: REAL;
	real_Multiplier_CH6: REAL;
	

			
END_VAR

//Creator : Stefan Lackner
//Company : EfficientIO
//Date : xx.09.2023
//Version : 1.0.0.0


//With this function is possible to read out all Information from a EL3446

//NOTE for diNr.....Designation => 
//_IN = Here Data come in from other Functions or go out to other functions about the GVL
//_OUT = Here Data go out to other functions about the GVL



(*-------------------------------------------------------------Service from Backend is ready and check the connection to backen for dissabel/enable Function---------------------------------------------------------------*)

//Try to reset the variable for connection on the GVL. When all is normal then the Lynus Mqtt connection function set this variable to true in the next cycle
//When we have no connection to the backend then after Lynus_Standards.Constants_General.tTimeDissableLynusFunctions days the Function is dissabled with all of his functionalities
timResetConnectionOnGVL(IN:= NOT timResetConnectionOnGVL.Q, PT:= T#1H, Q=> , ET=> );
IF timResetConnectionOnGVL.Q THEN 
	Lynus_Standards.GVL_Communicator.bStateConnectionToEnableFunctions := FALSE; 
END_IF
IF NOT Lynus_Standards.GVL_Communicator.bStateConnectionToEnableFunctions THEN 
	timDissableFunctions.IN := TRUE; 
ELSE 
	timDissableFunctions.IN := FALSE; 
END_IF  
timDissableFunctions(IN:= , PT:= Lynus_Standards.Constants_General.tTimeDissableLynusFunctions, Q=> , ET=> );

// limit inputs
uiCurrentTransformerRatio_CH1 := LIMIT (1,uiCurrentTransformerRatio_CH1,10000);
uiCurrentTransformerRatio_CH2 := LIMIT (1,uiCurrentTransformerRatio_CH2,10000);
uiCurrentTransformerRatio_CH3 := LIMIT (1,uiCurrentTransformerRatio_CH3,10000);
uiCurrentTransformerRatio_CH4 := LIMIT (1,uiCurrentTransformerRatio_CH4,10000);
uiCurrentTransformerRatio_CH5 := LIMIT (1,uiCurrentTransformerRatio_CH5,10000);
uiCurrentTransformerRatio_CH6 := LIMIT (1,uiCurrentTransformerRatio_CH6,10000);
uiVoltagePhaseSelector_CH1 := LIMIT (1,uiVoltagePhaseSelector_CH1,3);
uiVoltagePhaseSelector_CH2 := LIMIT (1,uiVoltagePhaseSelector_CH2,3);
uiVoltagePhaseSelector_CH3 := LIMIT (1,uiVoltagePhaseSelector_CH3,3);
uiVoltagePhaseSelector_CH4 := LIMIT (1,uiVoltagePhaseSelector_CH4,3);
uiVoltagePhaseSelector_CH5 := LIMIT (1,uiVoltagePhaseSelector_CH5,3);
uiVoltagePhaseSelector_CH6 := LIMIT (1,uiVoltagePhaseSelector_CH6,3);


(*----------------------------------------------------------------------------------------EL3446 Communication----------------------------------------------------------------------------------------------*)

// write CoE values for phase selector

IF 	NOT m_COE_Done OR uiVoltagePhaseSelector_CH1 <> uiVoltagePhaseSelector_old_CH1 OR uiVoltagePhaseSelector_CH2 <> uiVoltagePhaseSelector_old_CH2 OR
 	uiVoltagePhaseSelector_CH3 <> uiVoltagePhaseSelector_old_CH3 OR uiVoltagePhaseSelector_CH4 <> uiVoltagePhaseSelector_old_CH4 OR
  	uiVoltagePhaseSelector_CH5 <> uiVoltagePhaseSelector_old_CH5 OR uiVoltagePhaseSelector_CH6 <> uiVoltagePhaseSelector_old_CH6 
	THEN
	FB_CoE_EL3446.m_start := TRUE;
	m_COE_Done := TRUE;
	 uiVoltagePhaseSelector_old_CH1 := uiVoltagePhaseSelector_CH1;
	 uiVoltagePhaseSelector_old_CH2 := uiVoltagePhaseSelector_CH2;
	 uiVoltagePhaseSelector_old_CH3 := uiVoltagePhaseSelector_CH3;
	 uiVoltagePhaseSelector_old_CH4 := uiVoltagePhaseSelector_CH4;
	 uiVoltagePhaseSelector_old_CH5 := uiVoltagePhaseSelector_CH5;
	 uiVoltagePhaseSelector_old_CH6 := uiVoltagePhaseSelector_CH6;
END_IF
f_trig_Busy(CLK := FB_CoE_EL3446.m_Busy );
IF f_trig_Busy.Q AND (FB_CoE_EL3446.m_CoE_Write_done OR FB_CoE_EL3446.m_Error) THEN 
	FB_CoE_EL3446.m_start := FALSE;
END_IF
FB_CoE_EL3446(
	m_start:= , 
	nSlaveAddr:= nSlaveAddr,
	b_SubIndex:= b_SubIndex,
	uiVoltagePhaseSelector_CH1:= uiVoltagePhaseSelector_CH1, 
	uiVoltagePhaseSelector_CH2:= uiVoltagePhaseSelector_CH2, 
	uiVoltagePhaseSelector_CH3:= uiVoltagePhaseSelector_CH3, 
	uiVoltagePhaseSelector_CH4:= uiVoltagePhaseSelector_CH4, 
	uiVoltagePhaseSelector_CH5:= uiVoltagePhaseSelector_CH5, 
	uiVoltagePhaseSelector_CH6:= uiVoltagePhaseSelector_CH6, 
	m_Busy=> , 
	m_CoE_Write_done=> , 
	udint_GetAMSNetID_Error=> , 
	udint_WriteCoE_Error=> );

fbEL3446_wEL3443(
	bEnable:= TRUE, 
	pDpmData:= pDpmData, 
	stEL3446_IO:= , 
	stStatusPhase_I1=> , 
	stStatusPhase_I2=> , 
	stStatusPhase_I3=> , 
	stStatusPhase_I4=> , 
	stStatusPhase_I5=> , 
	stStatusPhase_I6=> , 
	stDPMVariantValues=> , 
	bError=> );
fbEL3446_wEL3443.stEL3446_IO.MDP5001_342_Input := stEL3446_IO.MDP5001_342_Input;
stEL3446_IO.MDP5001_342_Output := fbEL3446_wEL3443.stEL3446_IO.MDP5001_342_Output;
//Invert the Output data, because it is possible that the current transformers have been mounted in different mounting positions.
IF NOT bInvers_CH1 THEN
	real_Multiplier_CH1 := 1;
ELSE
	real_Multiplier_CH1 := -1;
END_IF
IF NOT bInvers_CH2 THEN
	real_Multiplier_CH2 := 1;
ELSE
	real_Multiplier_CH2 := -1;
END_IF
IF NOT bInvers_CH3 THEN
	real_Multiplier_CH3 := 1;
ELSE
	real_Multiplier_CH3 := -1;
END_IF
IF NOT bInvers_CH4 THEN
	real_Multiplier_CH4 := 1;
ELSE
	real_Multiplier_CH4 := -1;
END_IF
IF NOT bInvers_CH5 THEN
	real_Multiplier_CH5 := 1;
ELSE
	real_Multiplier_CH5 := -1;
END_IF
IF NOT bInvers_CH6 THEN
	real_Multiplier_CH6 := 1;
ELSE
	real_Multiplier_CH6 := -1;
END_IF

//Function
IF NOT bEnable3PhaseCH13 THEN
	fbEM_CH1(
		bEnable:= bEnable, 
		bError:= , 
		bEnableReadOutFunction:= FALSE, 
		bWriteWithDelay:= TRUE, 
		bPowerDataInvers:= FALSE,
		bReadOutDataDone:= timSetCounterValues.Q,
		iTimeReadOutInterval:= 0, 
		iErrorCode:= , 
		iWarningCode:= , 
		lrTotalCounterEnergy_Consumption:= fbEnergyCounter_CH1.lrTotalCounterEnergy_Consumption,
		lrTotalCounterEnergy_Production:= fbEnergyCounter_CH1.lrTotalCounterEnergy_Production, 
		lrCounterEnergyT1_Consumption:= fbEnergyCounter_CH1.lrCounterEnergyT1_Consumption,
		lrCounterEnergyT2_Consumption:= fbEnergyCounter_CH1.lrCounterEnergyT2_Consumption,
		lrCounterEnergyT1_Production:= fbEnergyCounter_CH1.lrCounterEnergyT1_Production, 
		lrCounterEnergyT2_Production:= fbEnergyCounter_CH1.lrCounterEnergyT2_Production, 
		lrCurrentL1:=  fbEL3446_wEL3443.stStatusPhase_I1.fCurrent * uiCurrentTransformerRatio_CH1,
		lrVoltageL1N:= , 
		lrVoltageL1L2:= , 
		lrPowerL1:= fbEL3446_wEL3443.stStatusPhase_I1.fActive_Power * uiCurrentTransformerRatio_CH1 * real_Multiplier_CH1, 
		lrCurrentL2:= ,
		lrVoltageL2N:= , 
		lrVoltageL2L3:= , 
		lrPowerL2:= , 
		lrCurrentL3:= , 
		lrVoltageL3N:= , 
		lrVoltageL3L1:= , 
		lrPowerL3:= , 
		lrPowerTotal:= fbEM_CH1.lrPowerL1, 
		lrFrequency:= stDataEMPowerRealTime.lrFrequency,  
		lrApparentPowerTotal:= fbEL3446_wEL3443.stStatusPhase_I1.fApparent_Power * uiCurrentTransformerRatio_CH1 ,
		lrReactivePowerTotal:= fbEL3446_wEL3443.stStatusPhase_I1.fReactive_Power_Fundamental * uiCurrentTransformerRatio_CH1, 
		tTimDelayOutput:= T#5S, 
		stDataEMOutPower=> stDataEMPowerRealTime_CH1, 
		stDataEMOutPowerDelay=> stDataEMPower_CH1, 
		stDataEMOutCounter=> stDataEMCounterRealTime_CH1,
		stDataEMOutCounterDelay=> stDataEMCounter_CH1,
		bReadOutMeter=> );
	fbEM_CH2(
		bEnable:= bEnable AND NOT timDissableFunctions.Q, 
		bError:= , 
		bEnableReadOutFunction:= FALSE, 
		bWriteWithDelay:= TRUE, 
		bPowerDataInvers:= FALSE,
		bReadOutDataDone:= timSetCounterValues.Q,
		iTimeReadOutInterval:= 0, 
		iErrorCode:= , 
		iWarningCode:= , 
		lrTotalCounterEnergy_Consumption:= fbEnergyCounter_CH2.lrTotalCounterEnergy_Consumption,
		lrTotalCounterEnergy_Production:= fbEnergyCounter_CH2.lrTotalCounterEnergy_Production, 
		lrCounterEnergyT1_Consumption:= fbEnergyCounter_CH2.lrCounterEnergyT1_Consumption,
		lrCounterEnergyT2_Consumption:= fbEnergyCounter_CH2.lrCounterEnergyT2_Consumption,
		lrCounterEnergyT1_Production:= fbEnergyCounter_CH2.lrCounterEnergyT1_Production, 
		lrCounterEnergyT2_Production:= fbEnergyCounter_CH2.lrCounterEnergyT2_Production, 
		lrCurrentL1:=  fbEL3446_wEL3443.stStatusPhase_I2.fCurrent * uiCurrentTransformerRatio_CH2,
		lrVoltageL1N:= , 
		lrVoltageL1L2:= , 
		lrPowerL1:= fbEL3446_wEL3443.stStatusPhase_I2.fActive_Power * uiCurrentTransformerRatio_CH2 * real_Multiplier_CH2, 
		lrCurrentL2:= ,
		lrVoltageL2N:= , 
		lrVoltageL2L3:= , 
		lrPowerL2:= , 
		lrCurrentL3:= , 
		lrVoltageL3N:= , 
		lrVoltageL3L1:= , 
		lrPowerL3:= , 
		lrPowerTotal:= fbEM_CH2.lrPowerL1, 
		lrFrequency:= stDataEMPowerRealTime.lrFrequency, 
		lrApparentPowerTotal:= fbEL3446_wEL3443.stStatusPhase_I2.fApparent_Power * uiCurrentTransformerRatio_CH2 ,
		lrReactivePowerTotal:= fbEL3446_wEL3443.stStatusPhase_I2.fReactive_Power_Fundamental * uiCurrentTransformerRatio_CH2, 
		tTimDelayOutput:= T#5S, 
		stDataEMOutPower=> stDataEMPowerRealTime_CH2, 
		stDataEMOutPowerDelay=> stDataEMPower_CH2, 
		stDataEMOutCounter=> stDataEMCounterRealTime_CH2,
		stDataEMOutCounterDelay=> stDataEMCounter_CH2,
		bReadOutMeter=> );
	fbEM_CH3(
		bEnable:= bEnable AND NOT timDissableFunctions.Q, 
		bError:= , 
		bEnableReadOutFunction:= FALSE, 
		bWriteWithDelay:= TRUE, 
		bPowerDataInvers:= FALSE,
		bReadOutDataDone:= timSetCounterValues.Q,
		iTimeReadOutInterval:= 0, 
		iErrorCode:= , 
		iWarningCode:= , 
		lrTotalCounterEnergy_Consumption:= fbEnergyCounter_CH3.lrTotalCounterEnergy_Consumption,
		lrTotalCounterEnergy_Production:= fbEnergyCounter_CH3.lrTotalCounterEnergy_Production, 
		lrCounterEnergyT1_Consumption:= fbEnergyCounter_CH3.lrCounterEnergyT1_Consumption,
		lrCounterEnergyT2_Consumption:= fbEnergyCounter_CH3.lrCounterEnergyT2_Consumption,
		lrCounterEnergyT1_Production:= fbEnergyCounter_CH3.lrCounterEnergyT1_Production, 
		lrCounterEnergyT2_Production:= fbEnergyCounter_CH3.lrCounterEnergyT2_Production, 
		lrCurrentL1:=  fbEL3446_wEL3443.stStatusPhase_I3.fCurrent * uiCurrentTransformerRatio_CH3,
		lrVoltageL1N:= , 
		lrVoltageL1L2:= , 
		lrPowerL1:= fbEL3446_wEL3443.stStatusPhase_I3.fActive_Power * uiCurrentTransformerRatio_CH3 * real_Multiplier_CH3, 
		lrCurrentL2:= ,
		lrVoltageL2N:= , 
		lrVoltageL2L3:= , 
		lrPowerL2:= , 
		lrCurrentL3:= , 
		lrVoltageL3N:= , 
		lrVoltageL3L1:= , 
		lrPowerL3:= , 
		lrPowerTotal:= fbEM_CH3.lrPowerL1, 
		lrFrequency:= stDataEMPowerRealTime.lrFrequency,
		lrApparentPowerTotal:= fbEL3446_wEL3443.stStatusPhase_I3.fApparent_Power * uiCurrentTransformerRatio_CH3 ,
		lrReactivePowerTotal:= fbEL3446_wEL3443.stStatusPhase_I3.fReactive_Power_Fundamental * uiCurrentTransformerRatio_CH3, 
		tTimDelayOutput:= T#5S, 
		stDataEMOutPower=> stDataEMPowerRealTime_CH3, 
		stDataEMOutPowerDelay=> stDataEMPower_CH3, 
		stDataEMOutCounter=> stDataEMCounterRealTime_CH3,
		stDataEMOutCounterDelay=> stDataEMCounter_CH3,
		bReadOutMeter=> );
	fbEnergyCounter_CH1(
		byActiveTariff:= 1, 
		lrPowerInput:= (fbEM_CH1.lrPowerL1) / 1000, 
		lrTotalCounterEnergy_Consumption=> , 
		lrTotalCounterEnergy_Production=> , 
		lrCounterEnergyT1_Consumption=> , 
		lrCounterEnergyT2_Consumption=> , 
		lrCounterEnergyT1_Production=> , 
		lrCounterEnergyT2_Production=> );
	fbEnergyCounter_CH2(
		byActiveTariff:= 1, 
		lrPowerInput:= (fbEM_CH2.lrPowerL1) / 1000, 
		lrTotalCounterEnergy_Consumption=> , 
		lrTotalCounterEnergy_Production=> , 
		lrCounterEnergyT1_Consumption=> , 
		lrCounterEnergyT2_Consumption=> , 
		lrCounterEnergyT1_Production=> , 
		lrCounterEnergyT2_Production=> );
	fbEnergyCounter_CH3(
		byActiveTariff:= 1, 
		lrPowerInput:= (fbEM_CH3.lrPowerL1) / 1000, 
		lrTotalCounterEnergy_Consumption=> , 
		lrTotalCounterEnergy_Production=> , 
		lrCounterEnergyT1_Consumption=> , 
		lrCounterEnergyT2_Consumption=> , 
		lrCounterEnergyT1_Production=> , 
		lrCounterEnergyT2_Production=> );
	CASE uiVoltagePhaseSelector_CH1 OF
		1: 	fbEM_CH1.lrVoltageL1N := stDataEMPowerRealTime.lrVoltageL1N;
		2: 	fbEM_CH1.lrVoltageL1N := stDataEMPowerRealTime.lrVoltageL2N;
		3: 	fbEM_CH1.lrVoltageL1N := stDataEMPowerRealTime.lrVoltageL3N;	
	END_CASE
	CASE uiVoltagePhaseSelector_CH2 OF
		1: 	fbEM_CH2.lrVoltageL1N := stDataEMPowerRealTime.lrVoltageL1N;
		2: 	fbEM_CH2.lrVoltageL1N := stDataEMPowerRealTime.lrVoltageL2N;
		3: 	fbEM_CH2.lrVoltageL1N := stDataEMPowerRealTime.lrVoltageL3N;	
	END_CASE
	CASE uiVoltagePhaseSelector_CH3 OF
		1: 	fbEM_CH3.lrVoltageL1N := stDataEMPowerRealTime.lrVoltageL1N;
		2: 	fbEM_CH3.lrVoltageL1N := stDataEMPowerRealTime.lrVoltageL2N;
		3: 	fbEM_CH3.lrVoltageL1N := stDataEMPowerRealTime.lrVoltageL3N;	
	END_CASE	
ELSE
	fbEM_CH1(
		bEnable:= bEnable AND NOT timDissableFunctions.Q, 
		bError:= , 
		bEnableReadOutFunction:= FALSE, 
		bWriteWithDelay:= TRUE, 
		bPowerDataInvers:= FALSE,
		bReadOutDataDone:= timSetCounterValues.Q,
		iTimeReadOutInterval:= 0, 
		iErrorCode:= , 
		iWarningCode:= , 
		lrTotalCounterEnergy_Consumption:= fbEnergyCounter_CH1.lrTotalCounterEnergy_Consumption,
		lrTotalCounterEnergy_Production:= fbEnergyCounter_CH1.lrTotalCounterEnergy_Production, 
		lrCounterEnergyT1_Consumption:= fbEnergyCounter_CH1.lrCounterEnergyT1_Consumption,
		lrCounterEnergyT2_Consumption:= fbEnergyCounter_CH1.lrCounterEnergyT2_Consumption,
		lrCounterEnergyT1_Production:= fbEnergyCounter_CH1.lrCounterEnergyT1_Production, 
		lrCounterEnergyT2_Production:= fbEnergyCounter_CH1.lrCounterEnergyT2_Production, 
		lrCurrentL1:=  fbEL3446_wEL3443.stStatusPhase_I1.fCurrent * uiCurrentTransformerRatio_CH1,
		lrVoltageL1N:= stDataEMPowerRealTime.lrVoltageL1N, 
		lrVoltageL1L2:= stDataEMPowerRealTime.lrVoltageL1L2, 
		lrPowerL1:= fbEL3446_wEL3443.stStatusPhase_I1.fActive_Power * uiCurrentTransformerRatio_CH1 * real_Multiplier_CH1, 
		lrCurrentL2:= fbEL3446_wEL3443.stStatusPhase_I2.fCurrent * uiCurrentTransformerRatio_CH2,
		lrVoltageL2N:= stDataEMPowerRealTime.lrVoltageL2N, 
		lrVoltageL2L3:=stDataEMPowerRealTime.lrVoltageL2L3 , 
		lrPowerL2:= fbEL3446_wEL3443.stStatusPhase_I2.fActive_Power * uiCurrentTransformerRatio_CH2 * real_Multiplier_CH2, 
		lrCurrentL3:=  fbEL3446_wEL3443.stStatusPhase_I3.fCurrent * uiCurrentTransformerRatio_CH3, 
		lrVoltageL3N:= stDataEMPowerRealTime.lrVoltageL3N, 
		lrVoltageL3L1:= stDataEMPowerRealTime.lrVoltageL3L1 , 
		lrPowerL3:= fbEL3446_wEL3443.stStatusPhase_I3.fActive_Power * uiCurrentTransformerRatio_CH3 * real_Multiplier_CH3, 
		lrPowerTotal:= fbEM_CH1.lrPowerL1 + fbEM_CH1.lrPowerL2 + fbEM_CH1.lrPowerL3,
		lrFrequency:= stDataEMPowerRealTime.lrFrequency, 
		lrApparentPowerTotal:= fbEL3446_wEL3443.stStatusPhase_I1.fApparent_Power * uiCurrentTransformerRatio_CH1 + fbEL3446_wEL3443.stStatusPhase_I2.fApparent_Power * uiCurrentTransformerRatio_CH2 + fbEL3446_wEL3443.stStatusPhase_I3.fApparent_Power * uiCurrentTransformerRatio_CH3,
		lrReactivePowerTotal:= fbEL3446_wEL3443.stStatusPhase_I1.fReactive_Power_Fundamental * uiCurrentTransformerRatio_CH1 + fbEL3446_wEL3443.stStatusPhase_I2.fReactive_Power_Fundamental * uiCurrentTransformerRatio_CH2 + fbEL3446_wEL3443.stStatusPhase_I3.fReactive_Power_Fundamental * uiCurrentTransformerRatio_CH3, 
		tTimDelayOutput:= T#5S, 
		stDataEMOutPower=> stDataEMPowerRealTime_CH1, 
		stDataEMOutPowerDelay=> stDataEMPower_CH1, 
		stDataEMOutCounter=> stDataEMCounterRealTime_CH1,
		stDataEMOutCounterDelay=> stDataEMCounter_CH1,
		bReadOutMeter=> );	
	fbEnergyCounter_CH1(
		byActiveTariff:= 1, 
		lrPowerInput:= (fbEM_CH1.lrPowerTotal) / 1000, 
		lrTotalCounterEnergy_Consumption=> , 
		lrTotalCounterEnergy_Production=> , 
		lrCounterEnergyT1_Consumption=> , 
		lrCounterEnergyT2_Consumption=> , 
		lrCounterEnergyT1_Production=> , 
		lrCounterEnergyT2_Production=> );
END_IF	
IF NOT bEnable3PhaseCH46 THEN 	
	fbEM_CH4(
		bEnable:= bEnable AND NOT timDissableFunctions.Q, 
		bError:= , 
		bEnableReadOutFunction:= FALSE, 
		bWriteWithDelay:= TRUE, 
		bPowerDataInvers:= FALSE,
		bReadOutDataDone:= timSetCounterValues.Q,
		iTimeReadOutInterval:= 0, 
		iErrorCode:= , 
		iWarningCode:= , 
		lrTotalCounterEnergy_Consumption:= fbEnergyCounter_CH4.lrTotalCounterEnergy_Consumption,
		lrTotalCounterEnergy_Production:= fbEnergyCounter_CH4.lrTotalCounterEnergy_Production, 
		lrCounterEnergyT1_Consumption:= fbEnergyCounter_CH4.lrCounterEnergyT1_Consumption,
		lrCounterEnergyT2_Consumption:= fbEnergyCounter_CH4.lrCounterEnergyT2_Consumption,
		lrCounterEnergyT1_Production:= fbEnergyCounter_CH4.lrCounterEnergyT1_Production, 
		lrCounterEnergyT2_Production:= fbEnergyCounter_CH4.lrCounterEnergyT2_Production, 
		lrCurrentL1:=  fbEL3446_wEL3443.stStatusPhase_I4.fCurrent * uiCurrentTransformerRatio_CH4,
		lrVoltageL1N:= , 
		lrVoltageL1L2:= , 
		lrPowerL1:= fbEL3446_wEL3443.stStatusPhase_I4.fActive_Power * uiCurrentTransformerRatio_CH4 * real_Multiplier_CH4, 
		lrCurrentL2:= ,
		lrVoltageL2N:= , 
		lrVoltageL2L3:= , 
		lrPowerL2:= , 
		lrCurrentL3:= , 
		lrVoltageL3N:= , 
		lrVoltageL3L1:= , 
		lrPowerL3:= , 
		lrPowerTotal:= fbEM_CH4.lrPowerL1, 
		lrFrequency:= stDataEMPowerRealTime.lrFrequency,
		lrApparentPowerTotal:= fbEL3446_wEL3443.stStatusPhase_I4.fApparent_Power * uiCurrentTransformerRatio_CH4 ,
		lrReactivePowerTotal:= fbEL3446_wEL3443.stStatusPhase_I4.fReactive_Power_Fundamental * uiCurrentTransformerRatio_CH4, 
		tTimDelayOutput:= T#5S, 
		stDataEMOutPower=> stDataEMPowerRealTime_CH4, 
		stDataEMOutPowerDelay=> stDataEMPower_CH4, 
		stDataEMOutCounter=> stDataEMCounterRealTime_CH4,
		stDataEMOutCounterDelay=> stDataEMCounter_CH4,
		bReadOutMeter=> );
	fbEM_CH5(
		bEnable:= bEnable AND NOT timDissableFunctions.Q, 
		bError:= , 
		bEnableReadOutFunction:= FALSE, 
		bWriteWithDelay:= TRUE, 
		bPowerDataInvers:= FALSE,
		bReadOutDataDone:= timSetCounterValues.Q,
		iTimeReadOutInterval:= 0, 
		iErrorCode:= , 
		iWarningCode:= , 
		lrTotalCounterEnergy_Consumption:= fbEnergyCounter_CH5.lrTotalCounterEnergy_Consumption,
		lrTotalCounterEnergy_Production:= fbEnergyCounter_CH5.lrTotalCounterEnergy_Production, 
		lrCounterEnergyT1_Consumption:= fbEnergyCounter_CH5.lrCounterEnergyT1_Consumption,
		lrCounterEnergyT2_Consumption:= fbEnergyCounter_CH5.lrCounterEnergyT2_Consumption,
		lrCounterEnergyT1_Production:= fbEnergyCounter_CH5.lrCounterEnergyT1_Production, 
		lrCounterEnergyT2_Production:= fbEnergyCounter_CH5.lrCounterEnergyT2_Production, 
		lrCurrentL1:=  fbEL3446_wEL3443.stStatusPhase_I5.fCurrent * uiCurrentTransformerRatio_CH5,
		lrVoltageL1N:= , 
		lrVoltageL1L2:= , 
		lrPowerL1:= fbEL3446_wEL3443.stStatusPhase_I5.fActive_Power * uiCurrentTransformerRatio_CH5 * real_Multiplier_CH5, 
		lrCurrentL2:= ,
		lrVoltageL2N:= , 
		lrVoltageL2L3:= , 
		lrPowerL2:= , 
		lrCurrentL3:= , 
		lrVoltageL3N:= , 
		lrVoltageL3L1:= , 
		lrPowerL3:= , 
		lrPowerTotal:= fbEM_CH5.lrPowerL1, 
		lrFrequency:= stDataEMPowerRealTime.lrFrequency,
		lrApparentPowerTotal:= fbEL3446_wEL3443.stStatusPhase_I5.fApparent_Power * uiCurrentTransformerRatio_CH5 ,
		lrReactivePowerTotal:= fbEL3446_wEL3443.stStatusPhase_I5.fReactive_Power_Fundamental * uiCurrentTransformerRatio_CH5, 
		tTimDelayOutput:= T#5S, 
		stDataEMOutPower=> stDataEMPowerRealTime_CH5, 
		stDataEMOutPowerDelay=> stDataEMPower_CH5, 
		stDataEMOutCounter=> stDataEMCounterRealTime_CH5,
		stDataEMOutCounterDelay=> stDataEMCounter_CH5,
		bReadOutMeter=> );
	fbEM_CH6(
		bEnable:= bEnable AND NOT timDissableFunctions.Q, 
		bError:= , 
		bEnableReadOutFunction:= FALSE, 
		bWriteWithDelay:= TRUE, 
		bPowerDataInvers:= FALSE,
		bReadOutDataDone:= timSetCounterValues.Q,
		iTimeReadOutInterval:= 0, 
		iErrorCode:= , 
		iWarningCode:= , 
		lrTotalCounterEnergy_Consumption:= fbEnergyCounter_CH6.lrTotalCounterEnergy_Consumption,
		lrTotalCounterEnergy_Production:= fbEnergyCounter_CH6.lrTotalCounterEnergy_Production, 
		lrCounterEnergyT1_Consumption:= fbEnergyCounter_CH6.lrCounterEnergyT1_Consumption,
		lrCounterEnergyT2_Consumption:= fbEnergyCounter_CH6.lrCounterEnergyT2_Consumption,
		lrCounterEnergyT1_Production:= fbEnergyCounter_CH6.lrCounterEnergyT1_Production, 
		lrCounterEnergyT2_Production:= fbEnergyCounter_CH6.lrCounterEnergyT2_Production, 
		lrCurrentL1:=  fbEL3446_wEL3443.stStatusPhase_I6.fCurrent * uiCurrentTransformerRatio_CH6,
		lrVoltageL1N:= , 
		lrVoltageL1L2:= , 
		lrPowerL1:= fbEL3446_wEL3443.stStatusPhase_I6.fActive_Power * uiCurrentTransformerRatio_CH6 * real_Multiplier_CH6, 
		lrCurrentL2:= ,
		lrVoltageL2N:= , 
		lrVoltageL2L3:= , 
		lrPowerL2:= , 
		lrCurrentL3:= , 
		lrVoltageL3N:= , 
		lrVoltageL3L1:= , 
		lrPowerL3:= , 
		lrPowerTotal:= fbEM_CH6.lrPowerL1, 
		lrFrequency:= stDataEMPowerRealTime.lrFrequency,
		lrApparentPowerTotal:= fbEL3446_wEL3443.stStatusPhase_I6.fApparent_Power * uiCurrentTransformerRatio_CH6 ,
		lrReactivePowerTotal:= fbEL3446_wEL3443.stStatusPhase_I6.fReactive_Power_Fundamental * uiCurrentTransformerRatio_CH6, 
		tTimDelayOutput:= T#5S, 
		stDataEMOutPower=> stDataEMPowerRealTime_CH6, 
		stDataEMOutPowerDelay=> stDataEMPower_CH6, 
		stDataEMOutCounter=> stDataEMCounterRealTime_CH6,
		stDataEMOutCounterDelay=> stDataEMCounter_CH6,
		bReadOutMeter=> );
	fbEnergyCounter_CH4(
		byActiveTariff:= 1, 
		lrPowerInput:= (fbEM_CH4.lrPowerL1) / 1000, 
		lrTotalCounterEnergy_Consumption=> , 
		lrTotalCounterEnergy_Production=> , 
		lrCounterEnergyT1_Consumption=> , 
		lrCounterEnergyT2_Consumption=> , 
		lrCounterEnergyT1_Production=> , 
		lrCounterEnergyT2_Production=> );
	fbEnergyCounter_CH5(
		byActiveTariff:= 1, 
		lrPowerInput:= (fbEM_CH5.lrPowerL1) / 1000, 
		lrTotalCounterEnergy_Consumption=> , 
		lrTotalCounterEnergy_Production=> , 
		lrCounterEnergyT1_Consumption=> , 
		lrCounterEnergyT2_Consumption=> , 
		lrCounterEnergyT1_Production=> , 
		lrCounterEnergyT2_Production=> );
	fbEnergyCounter_CH6(
		byActiveTariff:= 1, 
		lrPowerInput:= (fbEM_CH6.lrPowerL1) / 1000, 
		lrTotalCounterEnergy_Consumption=> , 
		lrTotalCounterEnergy_Production=> , 
		lrCounterEnergyT1_Consumption=> , 
		lrCounterEnergyT2_Consumption=> , 
		lrCounterEnergyT1_Production=> , 
		lrCounterEnergyT2_Production=> );
	CASE uiVoltagePhaseSelector_CH4 OF
		1: 	fbEM_CH4.lrVoltageL1N := stDataEMPowerRealTime.lrVoltageL1N;
		2: 	fbEM_CH4.lrVoltageL1N := stDataEMPowerRealTime.lrVoltageL2N;
		3: 	fbEM_CH4.lrVoltageL1N := stDataEMPowerRealTime.lrVoltageL3N;	
	END_CASE
	CASE uiVoltagePhaseSelector_CH5 OF
		1: 	fbEM_CH5.lrVoltageL1N := stDataEMPowerRealTime.lrVoltageL1N;
		2: 	fbEM_CH5.lrVoltageL1N := stDataEMPowerRealTime.lrVoltageL2N;
		3: 	fbEM_CH5.lrVoltageL1N := stDataEMPowerRealTime.lrVoltageL3N;	
	END_CASE
	CASE uiVoltagePhaseSelector_CH6 OF
		1: 	fbEM_CH6.lrVoltageL1N := stDataEMPowerRealTime.lrVoltageL1N;
		2: 	fbEM_CH6.lrVoltageL1N := stDataEMPowerRealTime.lrVoltageL2N;
		3: 	fbEM_CH6.lrVoltageL1N := stDataEMPowerRealTime.lrVoltageL3N;	
	END_CASE
ELSE 
	fbEM_CH4(
		bEnable:= bEnable AND NOT timDissableFunctions.Q, 
		bError:= , 
		bEnableReadOutFunction:= FALSE, 
		bWriteWithDelay:= TRUE, 
		bPowerDataInvers:= FALSE,
		bReadOutDataDone:= timSetCounterValues.Q,
		iTimeReadOutInterval:= 0, 
		iErrorCode:= , 
		iWarningCode:= , 
		lrTotalCounterEnergy_Consumption:= fbEnergyCounter_CH4.lrTotalCounterEnergy_Consumption,
		lrTotalCounterEnergy_Production:= fbEnergyCounter_CH4.lrTotalCounterEnergy_Production, 
		lrCounterEnergyT1_Consumption:= fbEnergyCounter_CH4.lrCounterEnergyT1_Consumption,
		lrCounterEnergyT2_Consumption:= fbEnergyCounter_CH4.lrCounterEnergyT2_Consumption,
		lrCounterEnergyT1_Production:= fbEnergyCounter_CH4.lrCounterEnergyT1_Production, 
		lrCounterEnergyT2_Production:= fbEnergyCounter_CH4.lrCounterEnergyT2_Production, 
		lrCurrentL1:=  fbEL3446_wEL3443.stStatusPhase_I4.fCurrent * uiCurrentTransformerRatio_CH4,
		lrVoltageL1N:= stDataEMPowerRealTime.lrVoltageL1N, 
		lrVoltageL1L2:= stDataEMPowerRealTime.lrVoltageL1L2, 
		lrPowerL1:= fbEL3446_wEL3443.stStatusPhase_I4.fActive_Power * uiCurrentTransformerRatio_CH4 * real_Multiplier_CH4, 
		lrCurrentL2:= fbEL3446_wEL3443.stStatusPhase_I5.fCurrent * uiCurrentTransformerRatio_CH5,
		lrVoltageL2N:= stDataEMPowerRealTime.lrVoltageL2N, 
		lrVoltageL2L3:=stDataEMPowerRealTime.lrVoltageL2L3 , 
		lrPowerL2:= fbEL3446_wEL3443.stStatusPhase_I5.fActive_Power * uiCurrentTransformerRatio_CH5 * real_Multiplier_CH5, 
		lrCurrentL3:=  fbEL3446_wEL3443.stStatusPhase_I6.fCurrent * uiCurrentTransformerRatio_CH6, 
		lrVoltageL3N:= stDataEMPowerRealTime.lrVoltageL3N, 
		lrVoltageL3L1:= stDataEMPowerRealTime.lrVoltageL3L1 , 
		lrPowerL3:= fbEL3446_wEL3443.stStatusPhase_I6.fActive_Power * uiCurrentTransformerRatio_CH6 * real_Multiplier_CH6, 
		lrPowerTotal:= fbEM_CH4.lrPowerL1 + fbEM_CH4.lrPowerL2 + fbEM_CH4.lrPowerL3,
		lrFrequency:= stDataEMPowerRealTime.lrFrequency, 
		lrApparentPowerTotal:= fbEL3446_wEL3443.stStatusPhase_I4.fApparent_Power * uiCurrentTransformerRatio_CH4 + fbEL3446_wEL3443.stStatusPhase_I5.fApparent_Power * uiCurrentTransformerRatio_CH5 + fbEL3446_wEL3443.stStatusPhase_I6.fApparent_Power * uiCurrentTransformerRatio_CH6,
		lrReactivePowerTotal:= fbEL3446_wEL3443.stStatusPhase_I4.fReactive_Power_Fundamental * uiCurrentTransformerRatio_CH4 + fbEL3446_wEL3443.stStatusPhase_I5.fReactive_Power_Fundamental * uiCurrentTransformerRatio_CH5 + fbEL3446_wEL3443.stStatusPhase_I6.fReactive_Power_Fundamental * uiCurrentTransformerRatio_CH6, 
		tTimDelayOutput:= T#5S, 
		stDataEMOutPower=> stDataEMPowerRealTime_CH4, 
		stDataEMOutPowerDelay=> stDataEMPower_CH4, 
		stDataEMOutCounter=> stDataEMCounterRealTime_CH4,
		stDataEMOutCounterDelay=> stDataEMCounter_CH4,
		bReadOutMeter=> );	
	fbEnergyCounter_CH4(
		byActiveTariff:= 1, 
		lrPowerInput:= (fbEM_CH4.lrPowerTotal) / 1000, 
		lrTotalCounterEnergy_Consumption=> , 
		lrTotalCounterEnergy_Production=> , 
		lrCounterEnergyT1_Consumption=> , 
		lrCounterEnergyT2_Consumption=> , 
		lrCounterEnergyT1_Production=> , 
		lrCounterEnergyT2_Production=> );
END_IF
(*----------------------------------------------------------------------------------------Electric Meter Function----------------------------------------------------------------------------------------------*)

//Error
IF timDissableFunctions.Q THEN 
	fbEM_CH1.bWarning := TRUE; 
	fbEM_CH1.iWarningCode := 0; 
ELSE 
	fbEM_CH1.bWarning := FALSE; 
END_IF 
IF Lynus_Standards.GVL_Energy.stNumberOfDevices.diNumberOfElectricMeters > Constants_Energy.diMaxNumberOfElectricMeters THEN 
	fbEM_CH1.bError := TRUE; 
ELSE 
	fbEM_CH1.bError := FALSE; 
END_IF
IF Lynus_Standards.GVL_Energy.stNumberOfDevices.diNumberOfElectricMeters > Constants_Energy.diMaxNumberOfElectricMeters THEN 
	fbEM_CH1.iErrorCode := 1;
ELSE 
	fbEM_CH1.iErrorCode := 0;
END_IF

timSetCounterValues(IN:= bEnable AND NOT timSetCounterValues.Q, PT:= T#2S, Q=> , ET=> );

END_FUNCTION_BLOCK

